METHOD SetDynConstraint_A : BOOL //Dynamic constraints for individual coordinates.
VAR_INPUT
    V : MC_LREAL; //equivalent to data type LREAL + MC_DEFAULT, MC_MAXIMUM
    A : MC_LREAL; //equivalent to data type LREAL + MC_DEFAULT, MC_MAXIMUM
    D : MC_LREAL; //equivalent to data type LREAL + MC_DEFAULT, MC_MAXIMUM
    J : MC_LREAL; //equivalent to data type LREAL + MC_DEFAULT, MC_MAXIMUM
END_VAR
THIS^.fbDynConstraintCoordinates.SetLimit(	Coordinate := Coord_Mcs_A1, 
											V := V, 
											A := A, 
											D := D, 
											J := J);
											
//Changes to the origin constraint do not affect the copy of the constraint in the instance of the DynamicConstraint_Container.
//For this reason, the container is being refreshed here							
fbDynConstraintContainer.Clear();
fbDynConstraintContainer.AddConstraint(fbDynConstraintPath);
fbDynConstraintContainer.AddConstraint(fbDynConstraintCoordinates);
END_METHOD

METHOD SetDynConstraint_B : BOOL //Dynamic constraints for individual coordinates.
VAR_INPUT
    V : MC_LREAL; //equivalent to data type LREAL + MC_DEFAULT, MC_MAXIMUM
    A : MC_LREAL; //equivalent to data type LREAL + MC_DEFAULT, MC_MAXIMUM
    D : MC_LREAL; //equivalent to data type LREAL + MC_DEFAULT, MC_MAXIMUM
    J : MC_LREAL; //equivalent to data type LREAL + MC_DEFAULT, MC_MAXIMUM
END_VAR
THIS^.fbDynConstraintCoordinates.SetLimit(	Coordinate := Coord_Mcs_B1, 
											V := V, 
											A := A, 
											D := D, 
											J := J);											

//Changes to the origin constraint do not affect the copy of the constraint in the instance of the DynamicConstraint_Container.
//For this reason, the container is being refreshed here							
fbDynConstraintContainer.Clear();
fbDynConstraintContainer.AddConstraint(fbDynConstraintPath);
fbDynConstraintContainer.AddConstraint(fbDynConstraintCoordinates);
END_METHOD

METHOD SetDynConstraint_C : BOOL //Dynamic constraints for individual coordinates.
VAR_INPUT
    V : MC_LREAL; //equivalent to data type LREAL + MC_DEFAULT, MC_MAXIMUM
    A : MC_LREAL; //equivalent to data type LREAL + MC_DEFAULT, MC_MAXIMUM
    D : MC_LREAL; //equivalent to data type LREAL + MC_DEFAULT, MC_MAXIMUM
    J : MC_LREAL; //equivalent to data type LREAL + MC_DEFAULT, MC_MAXIMUM
END_VAR
THIS^.fbDynConstraintCoordinates.SetLimit(	Coordinate := Coord_Mcs_C1, 
											V := V, 
											A := A, 
											D := D, 
											J := J);											

//Changes to the origin constraint do not affect the copy of the constraint in the instance of the DynamicConstraint_Container.
//For this reason, the container is being refreshed here							
fbDynConstraintContainer.Clear();
fbDynConstraintContainer.AddConstraint(fbDynConstraintPath);
fbDynConstraintContainer.AddConstraint(fbDynConstraintCoordinates);
END_METHOD

METHOD SetDynConstraint_Path : BOOL //One dimensional dynamic constraint along the XY-components of a path, ignoring non-tangential effects.
VAR_INPUT
    V : MC_LREAL; //equivalent to data type LREAL + MC_DEFAULT, MC_MAXIMUM
    A : MC_LREAL; //equivalent to data type LREAL + MC_DEFAULT, MC_MAXIMUM
    D : MC_LREAL; //equivalent to data type LREAL + MC_DEFAULT, MC_MAXIMUM
    J : MC_LREAL; //equivalent to data type LREAL + MC_DEFAULT, MC_MAXIMUM
END_VAR
THIS^.fbDynConstraintPath.SetValuesVADJ(V := V, 
										A := A, 
										D := D, 
										J := J);											

//Changes to the origin constraint do not affect the copy of the constraint in the instance of the DynamicConstraint_Container.
//For this reason, the container is being refreshed here							
fbDynConstraintContainer.Clear();
fbDynConstraintContainer.AddConstraint(fbDynConstraintPath);
fbDynConstraintContainer.AddConstraint(fbDynConstraintCoordinates);
END_METHOD

METHOD SetDynConstraint_X : BOOL //Dynamic constraints for individual coordinates.
VAR_INPUT
    V : MC_LREAL; //equivalent to data type LREAL + MC_DEFAULT, MC_MAXIMUM
    A : MC_LREAL; //equivalent to data type LREAL + MC_DEFAULT, MC_MAXIMUM
    D : MC_LREAL; //equivalent to data type LREAL + MC_DEFAULT, MC_MAXIMUM
    J : MC_LREAL; //equivalent to data type LREAL + MC_DEFAULT, MC_MAXIMUM
END_VAR
THIS^.fbDynConstraintCoordinates.SetLimit(	Coordinate := Coord_Mcs_X, 
											V := V, 
											A := A, 
											D := D, 
											J := J);											

//Changes to the origin constraint do not affect the copy of the constraint in the instance of the DynamicConstraint_Container.
//For this reason, the container is being refreshed here							
fbDynConstraintContainer.Clear();
fbDynConstraintContainer.AddConstraint(fbDynConstraintPath);
fbDynConstraintContainer.AddConstraint(fbDynConstraintCoordinates);
END_METHOD

METHOD SetDynConstraint_Y : BOOL //Dynamic constraints for individual coordinates.
VAR_INPUT
    V : MC_LREAL; //equivalent to data type LREAL + MC_DEFAULT, MC_MAXIMUM
    A : MC_LREAL; //equivalent to data type LREAL + MC_DEFAULT, MC_MAXIMUM
    D : MC_LREAL; //equivalent to data type LREAL + MC_DEFAULT, MC_MAXIMUM
    J : MC_LREAL; //equivalent to data type LREAL + MC_DEFAULT, MC_MAXIMUM
END_VAR
THIS^.fbDynConstraintCoordinates.SetLimit(	Coordinate := Coord_Mcs_Y, 
											V := V, 
											A := A, 
											D := D, 
											J := J);											

//Changes to the origin constraint do not affect the copy of the constraint in the instance of the DynamicConstraint_Container.
//For this reason, the container is being refreshed here							
fbDynConstraintContainer.Clear();
fbDynConstraintContainer.AddConstraint(fbDynConstraintPath);
fbDynConstraintContainer.AddConstraint(fbDynConstraintCoordinates);
END_METHOD

METHOD SetDynConstraint_Z : BOOL //Dynamic constraints for individual coordinates.
VAR_INPUT
    V : MC_LREAL; //equivalent to data type LREAL + MC_DEFAULT, MC_MAXIMUM
    A : MC_LREAL; //equivalent to data type LREAL + MC_DEFAULT, MC_MAXIMUM
    D : MC_LREAL; //equivalent to data type LREAL + MC_DEFAULT, MC_MAXIMUM
    J : MC_LREAL; //equivalent to data type LREAL + MC_DEFAULT, MC_MAXIMUM
END_VAR
THIS^.fbDynConstraintCoordinates.SetLimit(	Coordinate := Coord_Mcs_Z, 
											V := MC_DEFAULT, 
											A := A, 
											D := D, 
											J := J);											

//Changes to the origin constraint do not affect the copy of the constraint in the instance of the DynamicConstraint_Container.
//For this reason, the container is being refreshed here							
fbDynConstraintContainer.Clear();
fbDynConstraintContainer.AddConstraint(fbDynConstraintPath);
fbDynConstraintContainer.AddConstraint(fbDynConstraintCoordinates);
END_METHOD

METHOD Disable : HRESULT
VAR_INPUT
END_VAR
THIS^.eActiveCommand 				:= CHALET_NC.E_NcAxisCommands.Disable;
THIS^.fbFeedback.ActiveCommand 		:= TO_STRING(THIS^.eActiveCommand);	
THIS^.fbFeedback.LastCommandAccepted:= TRUE;		
THIS^.fbFeedback.Busy 				:= TRUE;

//Disable Axis
THIS^.fbMover.Disable(THIS^.fbFeedbackDisable);
Disable := S_OK;
END_METHOD

//This method is called when the system is disabled. Links are deleted as they may no longer be valid
METHOD Disassemble : HRESULT
VAR_INPUT
END_VAR

//Todo zzz Braucht es diese methode noch?
fbRouteComplete.Clear(); 
fbRouteRemaining.Clear(); 


Disassemble := S_OK;
END_METHOD

METHOD Enable : HRESULT
VAR_INPUT
END_VAR
IF NOT THIS^.fbFeedback.Busy THEN
	THIS^.eActiveCommand 				:= CHALET_NC.E_NcAxisCommands.Enable;
	THIS^.fbFeedback.ActiveCommand 		:= TO_STRING(THIS^.eActiveCommand);	
	THIS^.fbFeedback.LastCommandAccepted:= TRUE;		
	THIS^.fbFeedback.Busy 				:= TRUE;

	THIS^.fbMover.Enable(fbFeedbackEnable);
	Enable := S_OK;
ELSE
	Enable := S_FALSE;
	THIS^.fbFeedback.LastCommandAccepted:= FALSE;	
END_IF
END_METHOD

METHOD Reset : HRESULT
VAR_INPUT
END_VAR
THIS^.eActiveCommand 				:= CHALET_NC.E_NcAxisCommands.Reset;
THIS^.fbFeedback.ActiveCommand 		:= TO_STRING(THIS^.eActiveCommand);	
THIS^.fbFeedback.LastCommandAccepted:= TRUE;		
THIS^.fbFeedback.Busy 				:= TRUE;

THIS^.fbMover.Reset(THIS^.fbFeedbackReset);
Reset := S_OK;
END_METHOD

//Save the master mover and apply the distance traveled as a relative offset to this slave mover. Requires .StartExternalSetpoint()
METHOD AddMoverExtSetpoint : HRESULT
VAR_INPUT
	ipMasterMover : I_XP_Mover;
	fScalingX, fScalingY, fScalingZ, fScalingA, fScalingB, fScalingC : LREAL;// If >0, follow this axis to master-mover
END_VAR
//Invalide input
IF ipMasterMover = 0 THEN
	AddMoverExtSetpoint := E_FAIL;
	RETURN;
END_IF

//Allready stored a master
IF THIS^.ipMasterMover <> 0 THEN
	AddMoverExtSetpoint := E_FAIL;
	RETURN;
END_IF

//Only possible if ExternalSetpoint is not running
IF THIS^.nSeqStartExternalSetpoint <> 0 THEN
	AddMoverExtSetpoint := E_FAIL;
	RETURN;
END_IF



THIS^.ipMasterMover := ipMasterMover;
THIS^.stMasterMovementScaling.x := fScalingX;
THIS^.stMasterMovementScaling.y := fScalingy;
THIS^.stMasterMovementScaling.z := fScalingz;
THIS^.stMasterMovementScaling.a := fScalinga;
THIS^.stMasterMovementScaling.b := fScalingb;
THIS^.stMasterMovementScaling.c := fScalingc;
END_METHOD

{attribute 'monitoring':='call'}
PROPERTY  AxisExtSetpointA : CHALET_Nc.I_NcAxis_PLC
GET
AxisExtSetpointA := THIS^.AxisSetpointA;
END_GET
END_PROPERTY

{attribute 'monitoring':='call'}
PROPERTY AxisExtSetpointB : CHALET_Nc.I_NcAxis_PLC
GET
AxisExtSetpointB := THIS^.AxisSetpointB;
END_GET
END_PROPERTY

{attribute 'monitoring':='call'}
PROPERTY AxisExtSetpointC : CHALET_Nc.I_NcAxis_PLC
GET
AxisExtSetpointC := THIS^.AxisSetpointC;
END_GET
END_PROPERTY

{attribute 'monitoring':='call'}
PROPERTY  AxisExtSetpointX : CHALET_Nc.I_NcAxis_PLC
GET
AxisExtSetpointX := THIS^.AxisSetpointX;
END_GET
END_PROPERTY

{attribute 'monitoring':='call'}
PROPERTY AxisExtSetpointY : CHALET_Nc.I_NcAxis_PLC
GET
AxisExtSetpointY := THIS^.AxisSetpointY;
END_GET
END_PROPERTY

{attribute 'monitoring':='call'}
PROPERTY AxisExtSetpointZ : CHALET_Nc.I_NcAxis_PLC
GET
AxisExtSetpointZ := THIS^.AxisSetpointZ;
END_GET
END_PROPERTY

METHOD StartExternalSetpoint : HRESULT
THIS^.eActiveCommand 				:= CHALET_NC.E_NcAxisCommands.StartExternalSetpoint;
THIS^.fbFeedback.ActiveCommand 		:= TO_STRING(THIS^.eActiveCommand);		
THIS^.fbFeedback.Busy 				:= TRUE;


IF THIS^.fbMover.MCTOPLC.STD.State <> MC_PLANAR_STATE.Enabled THEN
	//Error wrong state
	
	;//zzz Todo Error message

ELSIF THIS^.bFeedExternalSetpointActive AND THIS^.nSeqStartExternalSetpoint = 999 THEN
	//Do nothing, setpoint is already active	
	THIS^.fbFeedbackExternalSetpointStartSeq.Done		:= TRUE;
	
ELSE
	
	//Start of internal sequence
	THIS^.fbFeedbackExternalSetpointStartSeq.Busy		:= TRUE;
	THIS^.nSeqStartExternalSetpoint := 1;
END_IF



StartExternalSetpoint := S_OK;
END_METHOD

METHOD StopExternalSetpoint : HRESULT
VAR_INPUT
END_VAR
AxisSetpointX.PowerOff();
AxisSetpointY.PowerOff();
AxisSetpointZ.PowerOff();
AxisSetpointA.PowerOff();
AxisSetpointB.PowerOff();
AxisSetpointC.PowerOff();


THIS^.eActiveCommand 				:= CHALET_NC.E_NcAxisCommands.StopExternalSetpoint;
THIS^.fbFeedback.ActiveCommand 		:= TO_STRING(THIS^.eActiveCommand);	
THIS^.fbFeedback.LastCommandAccepted:= TRUE;		


//Reset some flags
THIS^.nSeqStartExternalSetpoint := 0;
THIS^.bEvaluateFeedback := FALSE;
THIS^.ipMasterMover := 0;

IF THIS^.bFeedExternalSetpointActive THEN
	THIS^.fbMover.StopExternalSetpointGeneration(THIS^.fbFeedbackExtStop);	
	THIS^.bFeedExternalSetpointActive 	:= FALSE;
	THIS^.fbFeedback.Busy 				:= TRUE;
ELSE
	THIS^.fbFeedback.Done 				:= TRUE;
END_IF


StopExternalSetpoint := S_OK;
END_METHOD

METHOD PROTECTED UpdateExternalSetpoint : HRESULT
VAR
	SetPos, SetVelo, SetAcc : MoverVector;
	hr : HRESULT;
	stStartOptions : ST_ExternalSetpointGenerationOptions;
	stPosDifferenceToMasterMover : MoverVector;
	stPosOffsetMasterMover : MoverVector;
	stVeloOffsetMasterMover : MoverVector;
	stAccOffsetMasterMover : MoverVector;
END_VAR
IF NOT THIS^.Enabled THEN
	THIS^.nSeqStartExternalSetpoint := 0;
	THIS^.bFeedExternalSetpointActive := FALSE;
	THIS^.bEvaluateFeedback := FALSE;
END_IF


CASE nSeqStartExternalSetpoint OF
	0: //Wait for start
		;
		
	1: 	//store position of Master-Mover
		IF (THIS^.ipMasterMover <> 0) THEN
			THIS^.stMasterPositionAtStart := THIS^.ipMasterMover.PositionSet;
		END_IF

		//Reset all axis
		IF AxisSetpointX.Mapped THEN
			AxisSetpointX.Reset();
		END_IF
		IF AxisSetpointY.Mapped THEN
			AxisSetpointY.Reset();
		END_IF
		IF AxisSetpointZ.Mapped THEN
			AxisSetpointZ.Reset();
		END_IF
		IF AxisSetpointA.Mapped THEN
			AxisSetpointA.Reset();
		END_IF
		IF AxisSetpointB.Mapped THEN
			AxisSetpointB.Reset();
		END_IF
		IF AxisSetpointC.Mapped THEN
			AxisSetpointC.Reset();
		END_IF
		nSeqStartExternalSetpoint := nSeqStartExternalSetpoint + 1;		
		
		
	2: //Wait for feedback
		IF AxisSetpointX.Mapped THEN hr := GetMostSignificant(hr, AxisSetpointX.Feedback.HR); END_IF
		IF AxisSetpointY.Mapped THEN hr := GetMostSignificant(hr, AxisSetpointY.Feedback.HR); END_IF
		IF AxisSetpointZ.Mapped THEN hr := GetMostSignificant(hr, AxisSetpointZ.Feedback.HR); END_IF
		IF AxisSetpointA.Mapped THEN hr := GetMostSignificant(hr, AxisSetpointA.Feedback.HR); END_IF
		IF AxisSetpointB.Mapped THEN hr := GetMostSignificant(hr, AxisSetpointB.Feedback.HR); END_IF
		IF AxisSetpointC.Mapped THEN hr := GetMostSignificant(hr, AxisSetpointC.Feedback.HR); END_IF	
		IF hr = S_OK THEN
		 	nSeqStartExternalSetpoint := nSeqStartExternalSetpoint + 1;	
		END_IF
		
	3: 	//Reset all axis
		IF AxisSetpointX.Mapped THEN
			AxisSetpointX.PowerOn();
		END_IF
		IF AxisSetpointY.Mapped THEN
			AxisSetpointY.PowerOn();
		END_IF
		IF AxisSetpointZ.Mapped THEN
			AxisSetpointZ.PowerOn();
		END_IF
		IF AxisSetpointA.Mapped THEN
			AxisSetpointA.PowerOn();
		END_IF
		IF AxisSetpointB.Mapped THEN
			AxisSetpointB.PowerOn();
		END_IF
		IF AxisSetpointC.Mapped THEN
			AxisSetpointC.PowerOn();
		END_IF
		nSeqStartExternalSetpoint := nSeqStartExternalSetpoint + 1;		
		
	4: //Wait for feedback
		IF AxisSetpointX.Mapped THEN hr := GetMostSignificant(hr, AxisSetpointX.Feedback.HR); END_IF
		IF AxisSetpointY.Mapped THEN hr := GetMostSignificant(hr, AxisSetpointY.Feedback.HR); END_IF
		IF AxisSetpointZ.Mapped THEN hr := GetMostSignificant(hr, AxisSetpointZ.Feedback.HR); END_IF
		IF AxisSetpointA.Mapped THEN hr := GetMostSignificant(hr, AxisSetpointA.Feedback.HR); END_IF
		IF AxisSetpointB.Mapped THEN hr := GetMostSignificant(hr, AxisSetpointB.Feedback.HR); END_IF
		IF AxisSetpointC.Mapped THEN hr := GetMostSignificant(hr, AxisSetpointC.Feedback.HR); END_IF	
		IF hr = S_OK THEN
		 	nSeqStartExternalSetpoint := nSeqStartExternalSetpoint + 1;	
		END_IF

	5: 	//Enable all axis
		IF AxisSetpointX.Mapped THEN
			AxisSetpointX.SetActPosition(0.0);
		END_IF
		IF AxisSetpointY.Mapped THEN
			AxisSetpointY.SetActPosition(0.0);
		END_IF
		IF AxisSetpointZ.Mapped THEN
			AxisSetpointZ.SetActPosition(0.0);
		END_IF
		IF AxisSetpointA.Mapped THEN
			AxisSetpointA.SetActPosition(0.0);
		END_IF
		IF AxisSetpointB.Mapped THEN
			AxisSetpointB.SetActPosition(0.0);
		END_IF
		IF AxisSetpointC.Mapped THEN
			AxisSetpointC.SetActPosition(0.0);
		END_IF
		nSeqStartExternalSetpoint := nSeqStartExternalSetpoint + 1;		
		
	6: //Wait for feedback
		IF AxisSetpointX.Mapped THEN hr := GetMostSignificant(hr, AxisSetpointX.Feedback.HR); END_IF
		IF AxisSetpointY.Mapped THEN hr := GetMostSignificant(hr, AxisSetpointY.Feedback.HR); END_IF
		IF AxisSetpointZ.Mapped THEN hr := GetMostSignificant(hr, AxisSetpointZ.Feedback.HR); END_IF
		IF AxisSetpointA.Mapped THEN hr := GetMostSignificant(hr, AxisSetpointA.Feedback.HR); END_IF
		IF AxisSetpointB.Mapped THEN hr := GetMostSignificant(hr, AxisSetpointB.Feedback.HR); END_IF
		IF AxisSetpointC.Mapped THEN hr := GetMostSignificant(hr, AxisSetpointC.Feedback.HR); END_IF	
		IF hr = S_OK THEN
		 	nSeqStartExternalSetpoint := nSeqStartExternalSetpoint + 1;	
		END_IF

		
	7: // Activate external setpoint mode on mover
		stStartOptions.Mode := MC_EXTERNAL_SET_POSITION_MODE.Relative;
		THIS^.fbMover.StartExternalSetpointGeneration(	commandFeedback	:= THIS^.fbFeedbackExtStart,
														options 		:= stStartOptions);
		THIS^.bFeedExternalSetpointActive := TRUE;												
		nSeqStartExternalSetpoint := nSeqStartExternalSetpoint + 1;
	
		
	8: 
		THIS^.bEvaluateFeedback := TRUE;
		IF THIS^.fbFeedbackExtStart.Done THEN
			//Finish Sequence
			fbFeedbackExternalSetpointStartSeq.Done := TRUE;
			nSeqStartExternalSetpoint := 999;
		END_IF
		
	999: // finish seqence feedback
		
		
	1000..1999:
		//Error
		fbFeedbackExternalSetpointStartSeq.HR := E_FAIL;
END_CASE



IF THIS^.bFeedExternalSetpointActive THEN
	SetPos.X := AxisSetpointX.SetPosition;
	SetPos.Y := AxisSetpointY.SetPosition;
	SetPos.Z := AxisSetpointZ.SetPosition;
	SetPos.A := AxisSetpointA.SetPosition;
	SetPos.B := AxisSetpointB.SetPosition;
	SetPos.C := AxisSetpointC.SetPosition;
	
	SetVelo.X := AxisSetpointX.SetVelocity;
	SetVelo.Y := AxisSetpointY.SetVelocity;
	SetVelo.Z := AxisSetpointZ.SetVelocity;
	SetVelo.A := AxisSetpointA.SetVelocity;
	SetVelo.B := AxisSetpointB.SetVelocity;
	SetVelo.C := AxisSetpointC.SetVelocity;
	
	SetAcc.X := AxisSetpointX.SetAcceleration;
	SetAcc.Y := AxisSetpointY.SetAcceleration;
	SetAcc.Z := AxisSetpointZ.SetAcceleration;
	SetAcc.A := AxisSetpointA.SetAcceleration;
	SetAcc.B := AxisSetpointB.SetAcceleration;
	SetAcc.C := AxisSetpointC.SetAcceleration;
	
	IF THIS^.ipMasterMover <> 0 THEN
		//Difference to gearIn position
		stPosDifferenceToMasterMover := F_Vector_Subtraction(	minuend := THIS^.ipMasterMover.PositionSet, 
																subtrahend := stMasterPositionAtStart);
		//Add scaling factor	
		stPosOffsetMasterMover := F_Vector_Multiplication(	factor1 := stPosDifferenceToMasterMover,
															factor2 := THIS^.stMasterMovementScaling);							
		stVeloOffsetMasterMover := F_Vector_Multiplication(	factor1 := THIS^.ipMasterMover.VelocitySet,
															factor2 := THIS^.stMasterMovementScaling);							
		stAccOffsetMasterMover := F_Vector_Multiplication(	factor1 := THIS^.ipMasterMover.AccelerationSet,
															factor2 := THIS^.stMasterMovementScaling);						
		
		
		//Add Mastermover-Offest to 6-Axis-Offset
		SetPos := F_Vector_Addition( 	summand1 := stPosOffsetMasterMover,
									 	summand2 := SetPos);
		SetVelo := F_Vector_Addition( 	summand1 := stVeloOffsetMasterMover,
									 	summand2 := SetVelo);
		SetAcc := F_Vector_Addition( 	summand1 := stAccOffsetMasterMover,
									 	summand2 := SetAcc);
														
	END_IF
	
	//Send data to mover
	THIS^.fbMover.SetExternalSetpoint(	setPosition 		:= SetPos, 
										setVelocity 		:= SetVelo,
										setAcceleration 	:= SetAcc);
END_IF



CASE THIS^.eActiveCommand OF
	//Add the 6 axis to the feedback			
	E_NcAxisCommands.StartExternalSetpoint:
		//Only check MC_PlanarFeedback if cmd is active. Ignore old feedback
		IF THIS^.bEvaluateFeedback THEN
			fbFeedback.Busy 		:= fbFeedbackExtStart.Busy;
			fbFeedback.Done 		:= fbFeedbackExtStart.Done;
			fbFeedback.ErrorId 		:= fbFeedbackExtStart.ErrorID;
			fbFeedback.ClearObjectInfo();
		END_IF
		fbFeedback.HR := GetMostSignificant(fbFeedback.HR, fbFeedbackExternalSetpointStartSeq.HR);
		IF AxisSetpointX.Mapped THEN fbFeedback.HR := GetMostSignificant(fbFeedback.HR, AxisSetpointX.Feedback.HR);END_IF
		IF AxisSetpointY.Mapped THEN fbFeedback.HR := GetMostSignificant(fbFeedback.HR, AxisSetpointY.Feedback.HR);END_IF
		IF AxisSetpointZ.Mapped THEN fbFeedback.HR := GetMostSignificant(fbFeedback.HR, AxisSetpointZ.Feedback.HR);END_IF
		IF AxisSetpointA.Mapped THEN fbFeedback.HR := GetMostSignificant(fbFeedback.HR, AxisSetpointA.Feedback.HR);END_IF
		IF AxisSetpointB.Mapped THEN fbFeedback.HR := GetMostSignificant(fbFeedback.HR, AxisSetpointB.Feedback.HR);END_IF
		IF AxisSetpointC.Mapped THEN fbFeedback.HR := GetMostSignificant(fbFeedback.HR, AxisSetpointC.Feedback.HR);END_IF
		
	//Add the 6 axis to the feedback	
	E_NcAxisCommands.StopExternalSetpoint:
		fbFeedback.Busy 		:= fbFeedbackExtStop.Busy;
		fbFeedback.Done 		:= fbFeedbackExtStop.Done;
		fbFeedback.ErrorId 		:= fbFeedbackExtStop.ErrorID;
		fbFeedback.ClearObjectInfo(); 
		IF AxisSetpointX.Mapped THEN fbFeedback.HR := GetMostSignificant(fbFeedback.HR, AxisSetpointX.Feedback.HR);END_IF
		IF AxisSetpointY.Mapped THEN fbFeedback.HR := GetMostSignificant(fbFeedback.HR, AxisSetpointY.Feedback.HR);END_IF
		IF AxisSetpointZ.Mapped THEN fbFeedback.HR := GetMostSignificant(fbFeedback.HR, AxisSetpointZ.Feedback.HR);END_IF
		IF AxisSetpointA.Mapped THEN fbFeedback.HR := GetMostSignificant(fbFeedback.HR, AxisSetpointA.Feedback.HR);END_IF
		IF AxisSetpointB.Mapped THEN fbFeedback.HR := GetMostSignificant(fbFeedback.HR, AxisSetpointB.Feedback.HR);END_IF
		IF AxisSetpointC.Mapped THEN fbFeedback.HR := GetMostSignificant(fbFeedback.HR, AxisSetpointC.Feedback.HR);END_IF
END_CASE		


fbFeedbackExtStart.Update(); 
fbFeedbackExtStop.Update(); 


IF AxisSetpointX.Mapped THEN AxisSetpointX.Update() ;END_IF
IF AxisSetpointY.Mapped THEN AxisSetpointY.Update() ;END_IF
IF AxisSetpointZ.Mapped THEN AxisSetpointZ.Update() ;END_IF
IF AxisSetpointA.Mapped THEN AxisSetpointA.Update() ;END_IF
IF AxisSetpointB.Mapped THEN AxisSetpointB.Update() ;END_IF
IF AxisSetpointC.Mapped THEN AxisSetpointC.Update() ;END_IF
END_METHOD

METHOD AddToGroup : HRESULT
VAR_INPUT
	iGroup : I_XP_Group;
END_VAR
IF NOT THIS^.fbFeedback.Busy THEN
	THIS^.eActiveCommand 				:= CHALET_NC.E_NcAxisCommands.AddToGroupe;
	THIS^.fbFeedback.ActiveCommand 		:= TO_STRING(THIS^.eActiveCommand);	
	THIS^.fbFeedback.LastCommandAccepted:= TRUE;		
	THIS^.fbFeedback.Busy 				:= TRUE;
	
	iGroup.AddMover(THIS^.fbMover, THIS^.fbFeedbackAddToGrp);
	AddToGroup := S_OK;
ELSE
	AddToGroup := S_FALSE;
	THIS^.fbFeedback.LastCommandAccepted:= FALSE;	
END_IF
END_METHOD

METHOD RemoveFromGroup : HRESULT

VAR
	iGroup: INT;
END_VAR
IF NOT THIS^.fbFeedback.Busy THEN
	THIS^.eActiveCommand 				:= CHALET_NC.E_NcAxisCommands.RemoveFromGroupe;
	THIS^.fbFeedback.ActiveCommand 	:= TO_STRING(THIS^.eActiveCommand);	
	THIS^.fbFeedback.LastCommandAccepted:= TRUE;		
	THIS^.fbFeedback.Busy 				:= TRUE;
	
	THIS^.fbMover.RemoveFromGroup(THIS^.fbFeedbackRmvFromGrp);
	
	RemoveFromGroup := S_OK;
ELSE
	RemoveFromGroup := S_FALSE;
	THIS^.fbFeedback.LastCommandAccepted:= FALSE;	
END_IF
END_METHOD

//The mover returns to its SetPos. The force of the Z, A and B axis is slowly increased.
METHOD LiftFromUnknownLevel : HRESULT
VAR_INPUT
END_VAR
THIS^.eActiveCommand 				:= CHALET_NC.E_NcAxisCommands.LiftFromUnknownLevel;
THIS^.fbFeedback.ActiveCommand 		:= TO_STRING(THIS^.eActiveCommand);		
THIS^.fbFeedback.Busy 				:= TRUE;


IF THIS^.fbMover.MCTOPLC.STD.State <> MC_PLANAR_STATE.Enabled THEN
	//Error wrong state
	
	;//zzz Todo Error message
	
ELSIF NOT THIS^.Standstill THEN
	//Error not allowed if mover is moving
	
	;//zzz Todo Error message
	
ELSE
	//Start of internal sequence
	THIS^.fbFeedbackLiftFromUnknown.Busy		:= TRUE;
	THIS^.nSeqLiftFromUnknown := 1;
	THIS^.nSeqLowerToUnknown := 0;
END_IF



LiftFromUnknownLevel := S_OK;
END_METHOD

(* The mover is lowered. The target height is unknown. The force from the Z, A and B axles is then reduced to a minimum. X, Y and C still remain active.
   This function can be used, for example, to place the mover in a holder.  *)
METHOD LowerToUnknownLevel : HRESULT
VAR_INPUT
END_VAR
THIS^.eActiveCommand 				:= CHALET_NC.E_NcAxisCommands.LowerToUnknownLevel;
THIS^.fbFeedback.ActiveCommand 		:= TO_STRING(THIS^.eActiveCommand);		
THIS^.fbFeedback.Busy 				:= TRUE;


IF THIS^.fbMover.MCTOPLC.STD.State <> MC_PLANAR_STATE.Enabled THEN
	//Error wrong state
	
	;//zzz Todo Error message

ELSIF NOT THIS^.Standstill THEN
	//Error not allowed if mover is moving
	
	;//zzz Todo Error message
	
	
ELSE
	//Start of internal sequence
	THIS^.fbFeedbackLowerToUnknown.Busy		:= TRUE;
	THIS^.nSeqLowerToUnknown := 1;
	THIS^.nSeqLiftFromUnknown := 0;
END_IF



LowerToUnknownLevel := S_OK;
END_METHOD

METHOD PROTECTED UpdateUnknownLevel : HRESULT
VAR
	hr : HRESULT;
	stForceLimitMax: Tc3_XPlanarUtility.Force6D;
	stForceLimitMin: Tc3_XPlanarUtility.Force6D;
	stPosLagValueTemp : MoverVector;
	ipComObject: Tc3_Module.ITComObject;
	pstForcesAtBeginn : POINTER TO MoverVector;
END_VAR
VAR_INST
	fLowerNPerS : LREAL := 30.0;
	fLiftNPerS : LREAL := 50.0;
	fMaxForceFactor : LREAL := 1.0;
	fMinForceFactor : LREAL := 0.1;
	fPowerFactor : LREAL := 1.0;
	fCycleTime_s : LREAL; //[s]	
	bDoOnceIfDisabled : BOOL;
	stLagValuesAtBeginn : MoverVector;
	stForcesAtBeginn :  MoverVector;
	stForceLimitMaxAtBeginn : Tc3_XPlanarUtility.Force6D;
	stForceLimitMinAtBeginn : Tc3_XPlanarUtility.Force6D;
	stValideMinForce		: Tc3_XPlanarUtility.Force6D;
END_VAR
VAR CONSTANT
	N_PTCID_ForceLimitMax : PTCID := 16#03175051;
	N_PTCID_ForceLimitMin : PTCID := 16#03175052;
END_VAR
IF NOT THIS^.Enabled THEN
	THIS^.nSeqLowerToUnknown := 0;
	THIS^.nSeqLiftFromUnknown := 0;
	
	fCycleTime_s :=  TO_LREAL(TwinCAT_SystemInfoVarList._TaskInfo[THIS^.nTaskIndex].CycleTime(*100ns*)) / 10_000_000.0;
	stLagValuesAtBeginn := THIS^.UtilityMcMover.GetMaximumPositionLagValue();
END_IF

//if no TcIoMover is linked e.g. MC-Mover is in Simulation Mover:
IF THIS^.UtilityTcIoMover = 0 THEN
	IF fbFeedbackLowerToUnknown.Busy THEN
		fbFeedbackLowerToUnknown.Done := TRUE;
	END_IF
	IF fbFeedbackLiftFromUnknown.Busy THEN
		fbFeedbackLiftFromUnknown.Done := TRUE;
	END_IF
	RETURN;
END_IF



IF THIS^.ipXpSystem.Disabled AND bDoOnceIfDisabled THEN
	bDoOnceIfDisabled := FALSE;
	fPowerFactor := fMaxForceFactor;
	
	FW_ObjMgr_GetObjectInstance(oid:= THIS^.UtilityTcIoMover.ObjectId, iid:= TC_GLOBAL_IID_LIST.IID_ITComObject, pipUnk:= ADR(ipComObject));
	IF ipComObject <> 0 THEN
		// No minimum can be set if one of the 6 values in the struct is greater than the maximum. Equal is allowed.
		// The minimum is therefore first written to something valid. Followed by Max and the original minimum
		hr := ipComObject.TcSetObjPara(pid := N_PTCID_ForceLimitMin, nData := SIZEOF(stValideMinForce), pData := ADR(stValideMinForce), pgp := 0);
		hr := ipComObject.TcSetObjPara(pid := N_PTCID_ForceLimitMax, nData := SIZEOF(stForceLimitMaxAtBeginn), pData := ADR(stForceLimitMaxAtBeginn), pgp := 0);
		hr := ipComObject.TcSetObjPara(pid := N_PTCID_ForceLimitMin, nData := SIZEOF(stForceLimitMinAtBeginn), pData := ADR(stForceLimitMinAtBeginn), pgp := 0);
		FW_SafeRelease(ADR(ipComObject));
	END_IF

	THIS^.UtilityMcMover.SetMaximumPositionLagValue(stLagValuesAtBeginn);
END_IF


//Down
CASE nSeqLowerToUnknown OF
	0: //Wait for start
		;
		
	1: // Check if not already lewered	
		IF fPowerFactor = fMinForceFactor THEN
			nSeqLowerToUnknown := 999;
		ELSE
			nSeqLowerToUnknown := 5;
		END_IF
		
	5:	//Get some values
		pstForcesAtBeginn := THIS^.UtilityTcIoMover.ScopeAdr.GetOutputForce();
		stForcesAtBeginn := pstForcesAtBeginn^;
		stForceLimitMaxAtBeginn := THIS^.UtilityTcIoMover.GetForceLimitMax();
		stForceLimitMinAtBeginn := THIS^.UtilityTcIoMover.GetForceLimitMin();
		stValideMinForce.Fx := (stForceLimitMinAtBeginn.Fx * fMinForceFactor);
		stValideMinForce.Fy := (stForceLimitMinAtBeginn.Fy * fMinForceFactor);
		stValideMinForce.Fz := (stForceLimitMinAtBeginn.Fz * fMinForceFactor);
		stValideMinForce.Mx := (stForceLimitMinAtBeginn.Mx * fMinForceFactor);
		stValideMinForce.My := (stForceLimitMinAtBeginn.My * fMinForceFactor);
		stValideMinForce.Mz := (stForceLimitMinAtBeginn.Mz * fMinForceFactor);
		bDoOnceIfDisabled := TRUE;
		
		stPosLagValueTemp := stLagValuesAtBeginn;
		stPosLagValueTemp.z := THIS^.PositionSet.z + 0.5;
		THIS^.UtilityMcMover.SetMaximumPositionLagValue(stPosLagValueTemp);
		
		
		//0.0 - 1.0
		fPowerFactor := (stForcesAtBeginn.z / stForceLimitMaxAtBeginn.Fz);
		
		//add 5%
		fPowerFactor := fPowerFactor + 0.05;
		
		//Limit to 0.1 - 1.0
		fPowerFactor := MIN(fPowerFactor, fMaxForceFactor);
		fPowerFactor := MAX(fPowerFactor, fMinForceFactor);
		
		//set force Z, a and b
		stForceLimitMin := stForceLimitMinAtBeginn;		
		stForceLimitMin.fz := stForceLimitMin.Fz * fPowerFactor;
		stForceLimitMin.Mx := stForceLimitMin.Mx * fPowerFactor;
		stForceLimitMin.My := stForceLimitMin.My * fPowerFactor;
		
		stForceLimitMax := stForceLimitMaxAtBeginn;	
		stForceLimitMax.fz := stForceLimitMax.Fz * fPowerFactor;
		stForceLimitMax.Mx := stForceLimitMax.Mx * fPowerFactor;
		stForceLimitMax.My := stForceLimitMax.My * fPowerFactor;

		// 13.01.2025 Todo PLC Chash if Min > Max. use objParm insted
		//	THIS^.TcIoXPlanarMover.SetForceLimitMin(stForceLimitMin);
		//	THIS^.TcIoXPlanarMover.SetForceLimitMax(stForceLimitMax);
		FW_ObjMgr_GetObjectInstance(oid:= THIS^.UtilityTcIoMover.ObjectId, iid:= TC_GLOBAL_IID_LIST.IID_ITComObject, pipUnk:= ADR(ipComObject));
		IF ipComObject <> 0 THEN	
			// No minimum can be set if one of the 6 values in the struct is greater than the maximum. Equal is allowed.
			// The minimum is therefore first written to something valid. Followed by Max and the original minimum
			hr := ipComObject.TcSetObjPara(pid := N_PTCID_ForceLimitMin, nData := SIZEOF(stValideMinForce), pData := ADR(stValideMinForce), pgp := 0);
			hr := ipComObject.TcSetObjPara(pid := N_PTCID_ForceLimitMax, nData := SIZEOF(stForceLimitMax), pData := ADR(stForceLimitMax), pgp := 0);
			hr := ipComObject.TcSetObjPara(pid := N_PTCID_ForceLimitMin, nData := SIZEOF(stForceLimitMin), pData := ADR(stForceLimitMin), pgp := 0);
			FW_SafeRelease(ADR(ipComObject));
		END_IF

	
		nSeqLowerToUnknown := 10;
		
		
	10: 	
		//A lowering of the mover was detected followed by speed ~0
		IF (THIS^.PositionAct.z < THIS^.PositionSet.z * 0.5) AND (ABS(THIS^.VelocityAct.z) < 5.0)  THEN
			nSeqLowerToUnknown := 20;
			
		ELSIF (fPowerFactor <= fMinForceFactor) THEN
			nSeqLowerToUnknown := 20;
				
		ELSE
			//Reduce force each cycle
			fPowerFactor := fPowerFactor - ((fLowerNPerS/stForceLimitMaxAtBeginn.Fz) * fCycleTime_s);
					
			//Limit to 0.1 - 1.0
			fPowerFactor := MIN(fPowerFactor, fMaxForceFactor);
			fPowerFactor := MAX(fPowerFactor, fMinForceFactor);
			
			//set force Z, a and b to current + 10%
			stForceLimitMin := stForceLimitMinAtBeginn;		
			stForceLimitMin.fz := stForceLimitMin.Fz * fPowerFactor;
			stForceLimitMin.Mx := stForceLimitMin.Mx * fPowerFactor;
			stForceLimitMin.My := stForceLimitMin.My * fPowerFactor;
			
			stForceLimitMax := stForceLimitMaxAtBeginn;	
			stForceLimitMax.fz := stForceLimitMax.Fz * fPowerFactor;
			stForceLimitMax.Mx := stForceLimitMax.Mx * fPowerFactor;
			stForceLimitMax.My := stForceLimitMax.My * fPowerFactor;
	
			// 13.01.2025 Todo PLC Chash if Min > Max. use objParm insted
			//	THIS^.TcIoXPlanarMover.SetForceLimitMin(stForceLimitMin);
			//	THIS^.TcIoXPlanarMover.SetForceLimitMax(stForceLimitMax);
			FW_ObjMgr_GetObjectInstance(oid:= THIS^.UtilityTcIoMover.ObjectId, iid:= TC_GLOBAL_IID_LIST.IID_ITComObject, pipUnk:= ADR(ipComObject));
			IF ipComObject <> 0 THEN
				// No minimum can be set if one of the 6 values in the struct is greater than the maximum. Equal is allowed.
				// The minimum is therefore first written to something valid. Followed by Max and the original minimum
				hr := ipComObject.TcSetObjPara(pid := N_PTCID_ForceLimitMin, nData := SIZEOF(stValideMinForce), pData := ADR(stValideMinForce), pgp := 0);
				hr := ipComObject.TcSetObjPara(pid := N_PTCID_ForceLimitMax, nData := SIZEOF(stForceLimitMax), pData := ADR(stForceLimitMax), pgp := 0);
				hr := ipComObject.TcSetObjPara(pid := N_PTCID_ForceLimitMin, nData := SIZEOF(stForceLimitMin), pData := ADR(stForceLimitMin), pgp := 0);
				FW_SafeRelease(ADR(ipComObject));
			END_IF

	
		END_IF
	
		
	20: // Reduce Force to minimum
		fPowerFactor := fMinForceFactor;
		
		//set force Z, a and b to minimum
		stForceLimitMin := stForceLimitMinAtBeginn;		
		stForceLimitMin.fz := stForceLimitMin.Fz * fPowerFactor;
		stForceLimitMin.Mx := stForceLimitMin.Mx * fPowerFactor;
		stForceLimitMin.My := stForceLimitMin.My * fPowerFactor;
		
		stForceLimitMax := stForceLimitMaxAtBeginn;	
		stForceLimitMax.fz := stForceLimitMax.Fz * fPowerFactor;
		stForceLimitMax.Mx := stForceLimitMax.Mx * fPowerFactor;
		stForceLimitMax.My := stForceLimitMax.My * fPowerFactor;
	    
	    
		// 13.01.2025 Todo PLC Chash if Min > Max. use objParm insted
		//	THIS^.TcIoXPlanarMover.SetForceLimitMin(stForceLimitMin);
		//	THIS^.TcIoXPlanarMover.SetForceLimitMax(stForceLimitMax);
		FW_ObjMgr_GetObjectInstance(oid:= THIS^.UtilityTcIoMover.ObjectId, iid:= TC_GLOBAL_IID_LIST.IID_ITComObject, pipUnk:= ADR(ipComObject));
		IF ipComObject <> 0 THEN
			// No minimum can be set if one of the 6 values in the struct is greater than the maximum. Equal is allowed.
			// The minimum is therefore first written to something valid. Followed by Max and the original minimum
			hr := ipComObject.TcSetObjPara(pid := N_PTCID_ForceLimitMin, nData := SIZEOF(stValideMinForce), pData := ADR(stValideMinForce), pgp := 0);
			hr := ipComObject.TcSetObjPara(pid := N_PTCID_ForceLimitMax, nData := SIZEOF(stForceLimitMax), pData := ADR(stForceLimitMax), pgp := 0);
			hr := ipComObject.TcSetObjPara(pid := N_PTCID_ForceLimitMin, nData := SIZEOF(stForceLimitMin), pData := ADR(stForceLimitMin), pgp := 0);
			FW_SafeRelease(ADR(ipComObject));
		END_IF

		
		nSeqLowerToUnknown := 999;
				
	999: // finish seqence feedback
		fbFeedbackLowerToUnknown.Done := TRUE;
		
	1000..1999:
		//Error
		fbFeedbackLowerToUnknown.HR := E_FAIL;
END_CASE



//Up
CASE nSeqLiftFromUnknown OF
	0: //Wait for start
		;
		
	1: // Check if not already lifted	
		IF fPowerFactor = fMaxForceFactor THEN
			nSeqLiftFromUnknown := 999;
		ELSE
			nSeqLiftFromUnknown := 5;
		END_IF		
		
	5: 
		//0.0 - 1.0
		fPowerFactor := (stForcesAtBeginn.z / stForceLimitMaxAtBeginn.Fz);
		
		// -5%
		fPowerFactor := fPowerFactor - 0.05;
		
		//Limit to 0.1 - 1.0
		fPowerFactor := MIN(fPowerFactor, fMaxForceFactor);
		fPowerFactor := MAX(fPowerFactor, fMinForceFactor);
		
		//set force Z, a and b
		stForceLimitMin := stForceLimitMinAtBeginn;		
		stForceLimitMin.fz := stForceLimitMin.Fz * fPowerFactor;
		stForceLimitMin.Mx := stForceLimitMin.Mx * fPowerFactor;
		stForceLimitMin.My := stForceLimitMin.My * fPowerFactor;
		
		stForceLimitMax := stForceLimitMaxAtBeginn;	
		stForceLimitMax.fz := stForceLimitMax.Fz * fPowerFactor;
		stForceLimitMax.Mx := stForceLimitMax.Mx * fPowerFactor;
		stForceLimitMax.My := stForceLimitMax.My * fPowerFactor;

		// 13.01.2025 Todo PLC Chash if Min > Max. use objParm insted
		//THIS^.TcIoXPlanarMover.SetForceLimitMax(stForceLimitMax);
		//THIS^.TcIoXPlanarMover.SetForceLimitMin(stForceLimitMin);
		FW_ObjMgr_GetObjectInstance(oid:= THIS^.UtilityTcIoMover.ObjectId, iid:= TC_GLOBAL_IID_LIST.IID_ITComObject, pipUnk:= ADR(ipComObject));
		IF ipComObject <> 0 THEN
			// No minimum can be set if one of the 6 values in the struct is greater than the maximum. Equal is allowed.
			// The minimum is therefore first written to something valid. Followed by Max and the original minimum
			hr := ipComObject.TcSetObjPara(pid := N_PTCID_ForceLimitMin, nData := SIZEOF(stValideMinForce), pData := ADR(stValideMinForce), pgp := 0);
			hr := ipComObject.TcSetObjPara(pid := N_PTCID_ForceLimitMax, nData := SIZEOF(stForceLimitMax), pData := ADR(stForceLimitMax), pgp := 0);
			hr := ipComObject.TcSetObjPara(pid := N_PTCID_ForceLimitMin, nData := SIZEOF(stForceLimitMin), pData := ADR(stForceLimitMin), pgp := 0);
			FW_SafeRelease(ADR(ipComObject));
		END_IF
		
		nSeqLiftFromUnknown := 10;
		

		
	10: 	
		//A lift of the mover was detected followed by speed ~0
		IF (THIS^.PositionAct.z > THIS^.PositionSet.z * 0.5) AND (ABS(THIS^.VelocityAct.z) < 5.0)  THEN
			nSeqLiftFromUnknown := 20;
			
		ELSIF (fPowerFactor >= fMaxForceFactor ) THEN
			nSeqLiftFromUnknown := 20;
				
		ELSE
			//Reduce force each cycle
			fPowerFactor := fPowerFactor + ((fLiftNPerS/stForceLimitMaxAtBeginn.Fz) * fCycleTime_s);
					
			//Limit to 0.1 - 1.0
			fPowerFactor := MIN(fPowerFactor, fMaxForceFactor);
			fPowerFactor := MAX(fPowerFactor, fMinForceFactor);
			
			//set force Z, a and b 
			stForceLimitMin := stForceLimitMinAtBeginn;		
			stForceLimitMin.fz := stForceLimitMin.Fz * fPowerFactor;
			stForceLimitMin.Mx := stForceLimitMin.Mx * fPowerFactor;
			stForceLimitMin.My := stForceLimitMin.My * fPowerFactor;
			
			stForceLimitMax := stForceLimitMaxAtBeginn;	
			stForceLimitMax.fz := stForceLimitMax.Fz * fPowerFactor;
			stForceLimitMax.Mx := stForceLimitMax.Mx * fPowerFactor;
			stForceLimitMax.My := stForceLimitMax.My * fPowerFactor;
	
	
		// 13.01.2025 Todo PLC Chash if Min > Max. use objParm insted
		//THIS^.TcIoXPlanarMover.SetForceLimitMax(stForceLimitMax);
		//THIS^.TcIoXPlanarMover.SetForceLimitMin(stForceLimitMin);
		FW_ObjMgr_GetObjectInstance(oid:= THIS^.UtilityTcIoMover.ObjectId, iid:= TC_GLOBAL_IID_LIST.IID_ITComObject, pipUnk:= ADR(ipComObject));
		IF ipComObject <> 0 THEN
			// No minimum can be set if one of the 6 values in the struct is greater than the maximum. Equal is allowed.
			// The minimum is therefore first written to something valid. Followed by Max and the original minimum
			hr := ipComObject.TcSetObjPara(pid := N_PTCID_ForceLimitMin, nData := SIZEOF(stValideMinForce), pData := ADR(stValideMinForce), pgp := 0);
			hr := ipComObject.TcSetObjPara(pid := N_PTCID_ForceLimitMax, nData := SIZEOF(stForceLimitMax), pData := ADR(stForceLimitMax), pgp := 0);
			hr := ipComObject.TcSetObjPara(pid := N_PTCID_ForceLimitMin, nData := SIZEOF(stForceLimitMin), pData := ADR(stForceLimitMin), pgp := 0);
			FW_SafeRelease(ADR(ipComObject));
		END_IF
	
		END_IF
	
		
	20: // Reduce Force to normal			
		fPowerFactor := fMaxForceFactor;
		
		//set force Z, a and b to minimum
		stForceLimitMin := stForceLimitMinAtBeginn;		
		stForceLimitMin.fz := stForceLimitMin.Fz * fPowerFactor;
		stForceLimitMin.Mx := stForceLimitMin.Mx * fPowerFactor;
		stForceLimitMin.My := stForceLimitMin.My * fPowerFactor;
		
		stForceLimitMax := stForceLimitMaxAtBeginn;	
		stForceLimitMax.fz := stForceLimitMax.Fz * fPowerFactor;
		stForceLimitMax.Mx := stForceLimitMax.Mx * fPowerFactor;
		stForceLimitMax.My := stForceLimitMax.My * fPowerFactor;
	    	
		// 13.01.2025 Todo PLC Chash if Min > Max. use objParm insted
		//THIS^.TcIoXPlanarMover.SetForceLimitMax(stForceLimitMax);
		//THIS^.TcIoXPlanarMover.SetForceLimitMin(stForceLimitMin);
		FW_ObjMgr_GetObjectInstance(oid:= THIS^.UtilityTcIoMover.ObjectId, iid:= TC_GLOBAL_IID_LIST.IID_ITComObject, pipUnk:= ADR(ipComObject));
		IF ipComObject <> 0 THEN
			// No minimum can be set if one of the 6 values in the struct is greater than the maximum. Equal is allowed.
			// The minimum is therefore first written to something valid. Followed by Max and the original minimum
			hr := ipComObject.TcSetObjPara(pid := N_PTCID_ForceLimitMin, nData := SIZEOF(stValideMinForce), pData := ADR(stValideMinForce), pgp := 0);
			hr := ipComObject.TcSetObjPara(pid := N_PTCID_ForceLimitMax, nData := SIZEOF(stForceLimitMax), pData := ADR(stForceLimitMax), pgp := 0);
			hr := ipComObject.TcSetObjPara(pid := N_PTCID_ForceLimitMin, nData := SIZEOF(stForceLimitMin), pData := ADR(stForceLimitMin), pgp := 0);
			FW_SafeRelease(ADR(ipComObject));
		END_IF
		
		
		THIS^.UtilityMcMover.SetMaximumPositionLagValue(stLagValuesAtBeginn);
        
		nSeqLiftFromUnknown := 999;
				
	999: // finish seqence feedback
		fbFeedbackLiftFromUnknown.Done := TRUE;
		
	1000..1999:
		//Error
		fbFeedbackLiftFromUnknown.HR := E_FAIL;
END_CASE
END_METHOD

METHOD Halt : HRESULT
VAR_INPUT
END_VAR
THIS^.eActiveCommand 				:= CHALET_NC.E_NcAxisCommands.Halt;
THIS^.fbFeedback.ActiveCommand 		:= TO_STRING(THIS^.eActiveCommand);	
THIS^.fbFeedback.LastCommandAccepted:= TRUE;		
THIS^.fbFeedback.Busy 				:= TRUE;

THIS^.fbMover.Halt(	commandFeedback := THIS^.fbFeedbackHalt, 
					constraint 		:= THIS^.fbDynConstraintContainer 
				   );

Halt := S_OK;
END_METHOD

METHOD MoveA : HRESULT
VAR_INPUT
	fPosition : LREAL;
END_VAR
THIS^.eActiveCommand 				:= CHALET_NC.E_NcAxisCommands.MoveA;
THIS^.fbFeedback.ActiveCommand 		:= TO_STRING(THIS^.eActiveCommand);	
THIS^.fbFeedback.LastCommandAccepted:= TRUE;		
THIS^.fbFeedback.Busy 				:= TRUE;

THIS^.fbMover.MoveA(commandFeedback	:= THIS^.fbFeedbackMoveA, 
					targetPosition	:= fPosition, 
					constraint		:= THIS^.fbDynConstraintContainer
					);

MoveA := S_OK;
END_METHOD

METHOD MoveB : HRESULT
VAR_INPUT
	fPosition : LREAL;
END_VAR
THIS^.eActiveCommand 				:= CHALET_NC.E_NcAxisCommands.MoveB;
THIS^.fbFeedback.ActiveCommand 		:= TO_STRING(THIS^.eActiveCommand);	
THIS^.fbFeedback.LastCommandAccepted:= TRUE;		
THIS^.fbFeedback.Busy 				:= TRUE;

THIS^.fbMover.MoveB(commandFeedback	:= THIS^.fbFeedbackMoveB, 
					targetPosition	:= fPosition, 
					constraint		:= THIS^.fbDynConstraintContainer
					);

MoveB := S_OK;
END_METHOD

METHOD MoveC : HRESULT
VAR_INPUT
	fPosition : LREAL;
	
	(* Addition turns to move in modulo movement (positive or negative). *)
	additionalTurns : UDINT := 0;
	
	(* Direction in which the target is approached. *)
	direction : Tc3_Mc3Definitions.MC_DIRECTION := Tc3_Mc3Definitions.MC_DIRECTION.mcDirectionNonModulo;
END_VAR
VAR
	stMoveCOptions : ST_MoveCOptions;
END_VAR
THIS^.eActiveCommand 				:= CHALET_NC.E_NcAxisCommands.MoveC;
THIS^.fbFeedback.ActiveCommand 		:= TO_STRING(THIS^.eActiveCommand);	
THIS^.fbFeedback.LastCommandAccepted:= TRUE;		
THIS^.fbFeedback.Busy 				:= TRUE;


stMoveCOptions.additionalTurns := additionalTurns;
stMoveCOptions.direction := direction;


THIS^.fbMover.MoveC(commandFeedback	:= THIS^.fbFeedbackMoveC, 
					targetPosition	:= fPosition, 
					constraint		:= THIS^.fbDynConstraintContainer, 
					options			:= stMoveCOptions
					);

MoveC := S_OK;
END_METHOD

METHOD MoveXY : HRESULT
VAR_INPUT
	fPosition_X : LREAL;
	fPosition_Y : LREAL;
END_VAR
VAR
	fbTargetPosition 	: PositionXYC;
	stMoveOptions 		: ST_MoveToPositionOptions;
END_VAR
THIS^.eActiveCommand 				:= CHALET_NC.E_NcAxisCommands.MoveXY;
THIS^.fbFeedback.ActiveCommand 		:= TO_STRING(THIS^.eActiveCommand);	
THIS^.fbFeedback.LastCommandAccepted:= TRUE;		
THIS^.fbFeedback.Busy 				:= TRUE;



fbTargetPosition.SetValuesXY(x := fPosition_X, y := fPosition_Y);

stMoveOptions.useOrientation := TRUE;

THIS^.fbMover.MoveToPosition(	commandFeedback	:= THIS^.fbFeedbackMoveXY, 
								targetPosition	:= fbTargetPosition,
								constraint		:= THIS^.fbDynConstraintContainer, 
								options			:= stMoveOptions);

MoveXY := S_OK;
END_METHOD

METHOD MoveZ : HRESULT
VAR_INPUT
	fPosition : LREAL;
END_VAR
THIS^.eActiveCommand 				:= CHALET_NC.E_NcAxisCommands.MoveZ;
THIS^.fbFeedback.ActiveCommand 		:= TO_STRING(THIS^.eActiveCommand);	
THIS^.fbFeedback.LastCommandAccepted:= TRUE;		
THIS^.fbFeedback.Busy 				:= TRUE;


THIS^.fbMover.MoveZ(commandFeedback	:= THIS^.fbFeedbackMoveZ, 
					targetPosition	:= fPosition, 
					constraint		:= THIS^.fbDynConstraintContainer
					);

MoveZ := S_OK;
END_METHOD

{attribute 'monitoring':='call'}
(* Velocity is zero *)
PROPERTY Standstill : BOOL
GET
Standstill := TRUE;
Standstill := Standstill AND THIS^.PlanarMover.MCTOPLC.SET.SetVelo.x = 0;
Standstill := Standstill AND THIS^.PlanarMover.MCTOPLC.SET.SetVelo.y = 0;
Standstill := Standstill AND THIS^.PlanarMover.MCTOPLC.SET.SetVelo.z = 0;
Standstill := Standstill AND THIS^.PlanarMover.MCTOPLC.SET.SetVelo.a = 0;
Standstill := Standstill AND THIS^.PlanarMover.MCTOPLC.SET.SetVelo.b = 0;
Standstill := Standstill AND THIS^.PlanarMover.MCTOPLC.SET.SetVelo.c = 0;
END_GET
END_PROPERTY

{attribute 'monitoring':='call'}
//The last driving command given had the following value
PROPERTY LastCmdTargetGap : LREAL
GET
LastCmdTargetGap := fLastCmdTargetGap;
END_GET
END_PROPERTY

{attribute 'monitoring':='call'}
//The last driving command given had the following value
PROPERTY LastCmdTargetPosition : LREAL
GET
LastCmdTargetPosition := fLastCmdTargetPosition;
END_GET
END_PROPERTY

{attribute 'monitoring':='call'}
//The last driving command given had the following value
PROPERTY LastCmdTargetTrack: I_XP_Track
GET
LastCmdTargetTrack := ipLastCmdTrack;
END_GET
END_PROPERTY

{attribute 'monitoring':='call'}
//This was the last valid (system enabled) parent station of the mover
PROPERTY LastValidParentStation : I_XP_Station;
GET
VAR_INST

END_VAR
LastValidParentStation := THIS^.ipLastValidParentStation;
END_GET
END_PROPERTY

{attribute 'monitoring':='call'}
//This was the last valid (system enabled) actual  position of the mover
PROPERTY LastValidPositionOnTrack : LREAL
GET
VAR_INST

END_VAR
LastValidPositionOnTrack := THIS^.fLastValidPositionOnTrack;
END_GET
END_PROPERTY

{attribute 'monitoring':='call'}
//This was the last valid (system enabled) actual  position of the mover
PROPERTY LastValidPositionXYZABC : REFERENCE TO MoverVector
GET
VAR_INST

END_VAR
LastValidPositionXYZABC REF= THIS^.stLastValidPositionXYZABC;
END_GET
END_PROPERTY

{attribute 'monitoring':='call'}
//This was the last valid (system enabled) actual  position of the mover
PROPERTY LastValidTrack : I_XP_Track;
GET
VAR_INST

END_VAR
LastValidTrack := THIS^.ipLastValidTrack;
END_GET
END_PROPERTY

{attribute 'monitoring':='call'}
//Distance to the responsible parent station [mm]
PROPERTY DistToParentStation : LREAL
GET
VAR
	fDistToParentStationStartup : LREAL := CHALET_BaseComponents.GVL_Datatypes.cMaxLreal;
	fDistToParentStationReturn : LREAL;
	
	
	ipPath : I_XP_Path;
	bPathFound : BOOL;
	fTempDistToDest : LREAL;
	
	refPosOnTrack : REFERENCE TO MoverVector;
	ipNextWaypoint : I_XP_Station;
	
	fTotalLength : LREAL;
	fDistToBegin : LREAL;
END_VAR
IF THIS^.ParentStation = 0 THEN
	DistToParentStation := CHALET_BaseComponents.GVL_Datatypes.cMaxLreal;
	RETURN;
END_IF

//--- Not on track, line 
IF THIS^.CurrentTrack = 0 THEN
	refPosOnTrack REF= THIS^.ParentStation.PositionOnTrackXYZABC;
	fDistToParentStationReturn := F_DistXYVectors(THIS^.PositionAct,refPosOnTrack);
// ---- ---- ----	


//--- at startup there is no route - parent is station ahead
ELSIF THIS^.fbRouteComplete.IsEmpty THEN
	//check each path behind the parentstation if the mover is on it
	ParentStation.PathsBehinde.ResetIterator();
	WHILE ParentStation.PathsBehinde.HasNextObject() DO
		IF __QUERYINTERFACE(ParentStation.PathsBehinde.GetNextObject(), ipPath) THEN
			//get shortest distance
			fDistToParentStationStartup:= MIN(ipPath.DistanceToDestiantion(ipTrack:= THIS^.CurrentTrack, fPosOnTrack := THIS^.PositionOnTrack), fDistToParentStationStartup);
		END_IF
	END_WHILE
	ParentStation.PathsBehinde.RestoreIterator();	
	fDistToParentStationReturn := fDistToParentStationStartup;
// ---- ---- ----

// ---- Normal route dureing enabled system
ELSE
	THIS^.fbRouteComplete.ResetIterator();
	WHILE THIS^.fbRouteComplete.HasNextObject() DO
		IF __QUERYINTERFACE(THIS^.fbRouteComplete.GetNextObject(), ipPath) THEN
			fTotalLength := fTotalLength + ipPath.Length;
		
			IF NOT bPathFound THEN
				fTempDistToDest := ipPath.DistanceToDestiantion(ipTrack := THIS^.CurrentTrack, fPosOnTrack := THIS^.PositionOnTrack); 
				IF 	fTempDistToDest <> CHALET_BaseComponents.GVL_Datatypes.cMaxLreal THEN
					bPathFound := TRUE;
					fDistToParentStationReturn := fTempDistToDest;
				END_IF
			ELSE 
				fDistToParentStationReturn := fDistToParentStationReturn + ipPath.Length;
			END_IF
		END_IF
	END_WHILE
	THIS^.fbRouteComplete.RestoreIterator();
	// ---- ---- ----
	
	
	//--- If Mover is not on the path, return total length + dist to beginn
	IF NOT bPathFound THEN
		THIS^.fbRouteComplete.ResetIterator();
		IF __QUERYINTERFACE(THIS^.fbRouteComplete.GetNextObject(), ipPath) THEN
			refPosOnTrack REF= ipPath.StationDestination.PositionOnTrackXYZABC;
			fDistToBegin := F_DistXYVectors(THIS^.PositionAct, refPosOnTrack);	
		END_IF
		THIS^.fbRouteComplete.RestoreIterator();
		
		
		fDistToParentStationReturn := fDistToBegin + fTotalLength;
	END_IF
	 // ---- ---- ----

END_IF

DistToParentStation := fDistToParentStationReturn;

//Todo absturz, maximalwert von LREAL überschritten
//redce to 3 decimal places
//DistToParentStation := DINT_TO_LREAL(LREAL_TO_DINT(fDistToParentStationReturn*1000))/1000.0;
END_GET
END_PROPERTY

{attribute 'monitoring':='call'}
//Complete route from last parent to active parent station
PROPERTY RouteComplete : I_CH_List
GET
RouteComplete := THIS^.fbRouteComplete;
END_GET
END_PROPERTY

{attribute 'monitoring':='call'}
//Remaining route to the parent
PROPERTY RouteRemaining: I_CH_List
GET
RouteRemaining := THIS^.fbRouteRemaining;
END_GET
END_PROPERTY

//done segments can be transferred here. these are removed from the remaining route
METHOD RouteSegmentDone : BOOL
VAR_INPUT
	ipPathDone : I_XP_Path;
END_VAR
RouteSegmentDone := THIS^.fbRouteRemaining.RemoveObject(ipPathDone);
END_METHOD

METHOD SetRouteToParent : HRESULT
VAR_INPUT
	ipRoute : I_CH_LIST;
END_VAR
IF ipRoute = 0 THEN
	//Clear on empty input
	THIS^.fbRouteRemaining.Clear();
	THIS^.fbRouteComplete.Clear();
ELSE	
	//set as new route
	THIS^.fbRouteRemaining.Duplicate(ipRoute);
	THIS^.fbRouteComplete.Duplicate(ipRoute);	
END_IF
END_METHOD

{attribute 'monitoring':='call'}
(* Provides the current planar mover setpoint XYZABC [mm/s²] *)
PROPERTY AccelerationSet : REFERENCE TO MoverVector
GET
VAR_INST
	{attribute 'hide'}
	copyOfData :  MoverVector;
END_VAR
//Creat an copy of the struct to view value in targetdbrowser and plc online view
copyOfData := THIS^.fbMover.MCTOPLC.SET.SetAcc;
AccelerationSet REF= copyOfData;
END_GET
END_PROPERTY

{attribute 'monitoring':='call'}
(* C coordinate modulus set in MC3-Planar Mover[°] *)
PROPERTY CAxisModulo : LREAL
GET
VAR
	ipTrackComObject : ITComObject;
	nParaSize : UDINT;
	pParaData : PVOID;
	hr : HRESULT;
	fData : LREAL;
END_VAR
VAR CONSTANT
	N_IDX_OFFSET 	: UDINT := 16#05030107; // Parameter(init) Mover
END_VAR
FW_ObjMgr_GetObjectInstance(oid:= THIS^.OID, iid:= TC_GLOBAL_IID_LIST.IID_ITComObject, pipUnk:= ADR(ipTrackComObject));

IF ipTrackComObject = 0 THEN
	// Error
	RETURN;
END_IF


nParaSize := SIZEOF(fData);	pParaData := ADR(fData);

hr := ipTrackComObject.TcGetObjPara(pid:=N_IDX_OFFSET , nData:= nParaSize, pData:= pParaData, pgp:=0 );
FW_SafeRelease(ADR(ipTrackComObject));


CAxisModulo := TO_LREAL(TO_DINT(fData));
END_GET
END_PROPERTY

{attribute 'monitoring':='call'}
(* Indicates the command mode of an enabled PlanarMover, i.e. how setpoints are currently produced. *)
PROPERTY CommandMode : MC_PLANAR_MOVER_COMMAND_MODE
GET
CommandMode := THIS^.fbMover.MCTOPLC.STD.CommandMode;
END_GET
END_PROPERTY

{attribute 'monitoring':='call'}
//operational and position control active(hovering)
PROPERTY Enabled : BOOL
GET
(* StateDWord bit 20 - operational and position control active *)
Enabled :=  (THIS^.fbMover.MCTOPLC.STD.State = MC_PLANAR_STATE.Enabled) OR
			(THIS^.fbMover.MCTOPLC.STD.State = MC_PLANAR_STATE.Enabling) OR
			(THIS^.fbMover.MCTOPLC.STD.State = MC_PLANAR_STATE.Resetting AND PositionSet.z > 0.0) OR
			(THIS^.fbMover.MCTOPLC.STD.State = MC_PLANAR_STATE.Error AND PositionSet.z > 0.0) OR
			(THIS^.fbMover.MCTOPLC.STD.State = MC_PLANAR_STATE.ErrorPending AND PositionSet.z > 0.0) OR
			(THIS^.fbMover.MCTOPLC.STD.State = MC_PLANAR_STATE.Invalid AND PositionSet.z > 0.0);
END_GET
END_PROPERTY

{attribute 'monitoring':='call'}
(* Retruns lentgh of hypotenuse of the x and y error. (>=0[mm]) *)
PROPERTY LagDistanceXY : LREAL
GET
VAR
	fErrorX, fErrorY : LREAL;
END_VAR
// Set - Act
fErrorX := THIS^.fbMover.MCTOPLC.SET.SetPos.X - THIS^.fbMover.MCTOPLC.ACT.ActPos.X;
fErrorY := THIS^.fbMover.MCTOPLC.SET.SetPos.Y - THIS^.fbMover.MCTOPLC.ACT.ActPos.Y;


//Dist to center. Phytagoras -> c = sqrt( A^2 + B^2)
LagDistanceXY := SQRT(EXPT(fErrorX,2) + EXPT(fErrorY,2));
END_GET
END_PROPERTY

{attribute 'monitoring':='call'}
PROPERTY Mapped : BOOL //Project is mapped to MC (McToPlc and PlcToMc)
GET
VAR
	bMcToPlcNotMapped 	: BOOL;
	bPlcToMcNotMapped 	: BOOL;
END_VAR
//F_GetMappingStatus is not working on IO Data Pointer
	//bPlcToMcNotMapped := F_GetMappingStatus(ADR(THIS^.fbMover.PlcToMc), SIZEOF(THIS^.fbMover.PlcToMc)) <> EPlcMappingStatus.MS_Mapped;
	//bMcToPlcNotMapped := F_GetMappingStatus(ADR(THIS^.fbMover.McToPlc), SIZEOF(THIS^.fbMover.McToPlc)) <> EPlcMappingStatus.MS_Mapped;

	
Mapped := THIS^.fbMover.MCTOPLC.STD.MoverOID <> 0;
END_GET
END_PROPERTY

{attribute 'monitoring':='call'}
PROPERTY Mode : MC_PLANAR_MOVER_COMMAND_MODE
GET
Mode := THIS^.fbMover.MCTOPLC.STD.CommandMode;
END_GET
END_PROPERTY

{attribute 'monitoring':='call'}
(* Height that is used for internal collision checks.[mm] *)
PROPERTY MoverHeight : LREAL
GET
VAR
	ipTrackComObject : ITComObject;
	nParaSize : UDINT;
	pParaData : PVOID;
	hr : HRESULT;
	fData : LREAL;
END_VAR
VAR CONSTANT
	N_IDX_OFFSET 	: UDINT := 16#050300B3; // Parameter(init) Mover
END_VAR
FW_ObjMgr_GetObjectInstance(oid:= THIS^.OID, iid:= TC_GLOBAL_IID_LIST.IID_ITComObject, pipUnk:= ADR(ipTrackComObject));

IF ipTrackComObject = 0 THEN
	// Error
	RETURN;
END_IF


nParaSize := SIZEOF(fData);	pParaData := ADR(fData);

hr := ipTrackComObject.TcGetObjPara(pid:=N_IDX_OFFSET , nData:= nParaSize, pData:= pParaData, pgp:=0 );
FW_SafeRelease(ADR(ipTrackComObject));


MoverHeight := fData;
END_GET
END_PROPERTY

{attribute 'monitoring':='call'}
//Mover could not be detected or was removed from the system
PROPERTY MoverIsNotPresent : BOOL
GET
VAR
	bMoverAtZeroPos, bMoverPositionInvalid, bMoverVeloInvalid : BOOL;
END_VAR
bMoverAtZeroPos		:=  PlanarMover.MCTOPLC.ACT.ActPos.x = 0 AND
						PlanarMover.MCTOPLC.ACT.ActPos.y = 0 AND 
						PlanarMover.MCTOPLC.ACT.ActPos.z = 0 AND 
						PlanarMover.MCTOPLC.ACT.ActPos.a = 0 AND
						PlanarMover.MCTOPLC.ACT.ActPos.b = 0 AND 
						PlanarMover.MCTOPLC.ACT.ActPos.c = 0 AND 
						PlanarMover.MCTOPLC.ACT.PhysicalAreaID = 0;
						
						
bMoverPositionInvalid:=  PlanarMover.MCTOPLC.ACT.ActPos.x >= 1E+302 AND
						PlanarMover.MCTOPLC.ACT.ActPos.y >= 1E+302 AND 
						PlanarMover.MCTOPLC.ACT.ActPos.z >= 1E+302 AND 
						PlanarMover.MCTOPLC.ACT.ActPos.a >= 1E+302 AND
						PlanarMover.MCTOPLC.ACT.ActPos.b >= 1E+302 AND 
						PlanarMover.MCTOPLC.ACT.ActPos.c >= 1E+302;
						
						
bMoverVeloInvalid	:=  PlanarMover.MCTOPLC.ACT.ActVelo.x >= 1E+302 AND
						PlanarMover.MCTOPLC.ACT.ActVelo.y >= 1E+302 AND 
						PlanarMover.MCTOPLC.ACT.ActVelo.z >= 1E+302 AND 
						PlanarMover.MCTOPLC.ACT.ActVelo.a >= 1E+302 AND
						PlanarMover.MCTOPLC.ACT.ActVelo.b >= 1E+302 AND 
						PlanarMover.MCTOPLC.ACT.ActVelo.c >= 1E+302;
						
MoverIsNotPresent := bMoverAtZeroPos OR bMoverPositionInvalid OR bMoverVeloInvalid;
END_GET
END_PROPERTY

{attribute 'monitoring':='call'}
(* Width that is used for internal collision checks.[mm] *)
PROPERTY MoverWidth : LREAL
GET
VAR
	ipTrackComObject : ITComObject;
	nParaSize : UDINT;
	pParaData : PVOID;
	hr : HRESULT;
	fData : LREAL;
END_VAR
VAR CONSTANT
	N_IDX_OFFSET 	: UDINT := 16#050300B2; // Parameter(init) Mover
END_VAR
FW_ObjMgr_GetObjectInstance(oid:= THIS^.OID, iid:= TC_GLOBAL_IID_LIST.IID_ITComObject, pipUnk:= ADR(ipTrackComObject));

IF ipTrackComObject = 0 THEN
	// Error
	RETURN;
END_IF


nParaSize := SIZEOF(fData);	pParaData := ADR(fData);
hr := ipTrackComObject.TcGetObjPara(pid:=N_IDX_OFFSET , nData:= nParaSize, pData:= pParaData, pgp:=0 );
FW_SafeRelease(ADR(ipTrackComObject));

MoverWidth := fData;
END_GET
END_PROPERTY

{attribute 'monitoring':='call'}
(* Contains the information of the Planar Mover passed from MC to PLC. XYZABC [mm] *)
PROPERTY PositionAct : REFERENCE TO MoverVector
GET
VAR_INST
	{attribute 'hide'}
	copyOfActPosition :  MoverVector;
END_VAR
//Creat an copy of the struct to view value in targetdbrowser and plc online view
copyOfActPosition := THIS^.fbMover.MCTOPLC.ACT.ActPos;
PositionAct REF= copyOfActPosition;
END_GET
END_PROPERTY

{attribute 'monitoring':='call'}
(* Provides the current planar mover setpoint XYZABC [mm] *)
PROPERTY PositionSet : REFERENCE TO MoverVector
GET
VAR_INST
	{attribute 'hide'}
	copyOfSetPosition :  MoverVector;
END_VAR
//Creat an copy of the struct to view value in targetdbrowser and plc online view
copyOfSetPosition := THIS^.fbMover.MCTOPLC.SET.SetPos;
PositionSet REF= copyOfSetPosition;
END_GET
END_PROPERTY

{attribute 'monitoring':='call'}
PROPERTY PUBLIC ProductData : I_XP_ProductData
GET
ProductData := ipProductData;
END_GET
SET
// No change. Same interface is set again
IF ipProductData = ProductData THEN
	;//Noting
	
ELSE

	// If allready an interface is linked. Unlink
	IF ipProductData <> 0 THEN
		ipProductData.LinkToMover(0);
		ipProductData := 0;
	END_IF
	
	// Link and store new interface
	IF ProductData <> 0 THEN
		ProductData.LinkToMover(THIS^);
		ipProductData := ProductData;
	END_IF
END_IF
END_SET
END_PROPERTY

{attribute 'monitoring':='call'}
(* Provides the current planar mover act XYZABC [mm/s] *)
PROPERTY VelocityAct : REFERENCE TO MoverVector
GET
VAR_INST
	{attribute 'hide'}
	copyOfData :  MoverVector;
END_VAR
//Creat an copy of the struct to view value in targetdbrowser and plc online view
copyOfData := THIS^.fbMover.MCTOPLC.ACT.ActVelo;
VelocityAct REF= copyOfData;
END_GET
END_PROPERTY

{attribute 'monitoring':='call'}
(* Provides the current planar mover setpoint XYZABC [mm/s] *)
PROPERTY VelocitySet : REFERENCE TO MoverVector
GET
VAR_INST
	{attribute 'hide'}
	copyOfData :  MoverVector;
END_VAR
//Creat an copy of the struct to view value in targetdbrowser and plc online view
copyOfData := THIS^.fbMover.MCTOPLC.SET.SetVelo;
VelocitySet REF= copyOfData;
END_GET
END_PROPERTY

{attribute 'monitoring':='call'}
PROPERTY CurrentTrack : I_XP_Track
GET
VAR
	ipTrackObj : I_CH_Object;
	ipTrack : I_XP_Track;
END_VAR
IF ipXpSystem <> 0 THEN
	ipTrackObj := ipXpSystem.Tracks.FindOID(THIS^.PlanarMover.MCTOPLC.SETONTRACK.TrackOID);
	ToXpTrack(ipTrackObj,ipTrack);
END_IF

CurrentTrack := ipTrack;
END_GET
END_PROPERTY

METHOD DistToTrack : LREAL
VAR_INPUT
	iTrack : I_XP_Track;
END_VAR
VAR
	fPositionOnTrack : LREAL;
	trackPosition, moverPosition : PositionXYC;
END_VAR
moverPosition.x := PositionSet.x;
moverPosition.y := PositionSet.y;
moverPosition.c := PositionSet.c;

//Get Pos on track in mm
fPositionOnTrack := iTrack.PlanarTrack.GetArcLengthClosestTo(geometry:=moverPosition);

//Convert pos on track in XY
iTrack.PlanarTrack.GetPositionAt(arcLength := fPositionOnTrack, position:=trackPosition);

//Get distance to mover
DistToTrack := SQRT(EXPT((trackPosition.x - moverPosition.x),2)+EXPT((trackPosition.y - moverPosition.y),2));
END_METHOD

METHOD JoinTrack : HRESULT
VAR_INPUT
	iTrack : I_XP_Track;
END_VAR
VAR
	joinTrackOptions : ST_JoinTrackOptions;
END_VAR
IF iTrack <> 0 THEN
	THIS^.eActiveCommand 				:= CHALET_NC.E_NcAxisCommands.JoinTrack;
	THIS^.fbFeedback.ActiveCommand 		:= TO_STRING(THIS^.eActiveCommand);	
	THIS^.fbFeedback.LastCommandAccepted:= TRUE;		
	THIS^.fbFeedback.Busy 				:= TRUE;

	
	(* ADS Error 33164 or 33154: Position out of modulo range or Software position limit violation. Position must be larger or equal to zero and less or equal to the modulus when using modulo positioning. 
		When using modulo positioning, the target position is interpreted in consideration of the AdditionalTurns variable at the Options input.

		If the above error occurs, then the mover wants to rotate on the track when joining because ‘useOrientation = TRUE’ is set. 
		Better do not to set this to false, because CA then requires a much greater distance to the neighbouring mover.
		It is better to check the set C-axis modules in the MC3 PlanarMover if 90, 180 or 360°.
	*)
	joinTrackOptions.useOrientation 	:= TRUE;

	
	THIS^.fbMover.JoinTrack(commandFeedback	:= THIS^.fbFeedbackJoinTrack, 
								targetTrack	:= iTrack.PlanarTrack, 
								constraint	:= THIS^.fbDynConstraintContainer,
								options		:= joinTrackOptions);								
	JoinTrack := S_OK;
ELSE
	JoinTrack := S_FALSE;
	THIS^.fbFeedback.LastCommandAccepted:= FALSE;	
END_IF
END_METHOD

METHOD MoveOnTrack : HRESULT
VAR_INPUT
	ipTrack : I_XP_Track;
	fPosition : LREAL;
	fGap : LREAL;
END_VAR

VAR
	moveOptions: ST_MoveOnTrackOptions;
	//fMoverDiagonal : LREAL;
END_VAR
moveOptions.direction := Tc3_Mc3Definitions.MC_DIRECTION.mcDirectionPositive;
moveOptions.additionalTurns := 0;
moveOptions.gap := XPlanarParameterlist.N_GAP_MODE_ON_TRACK; 

//Use fix gap if requested gap is to small
moveOptions.gap := MAX(fGap, XPlanarParameterlist.F_MOVER_MINIMUM_GAP_ON_TRACK);
moveOptions.dynamicMode := XPlanarParameterlist.N_SELECT_MODE_HOW_DYNAMIC_IS_PLANED_ON_TRACK;

IF ipTrack <> 0 THEN
	THIS^.eActiveCommand 				:= CHALET_NC.E_NcAxisCommands.MoveOnTrack;
	THIS^.fbFeedback.ActiveCommand 		:= TO_STRING(THIS^.eActiveCommand);	
	THIS^.fbFeedback.LastCommandAccepted:= TRUE;		
	THIS^.fbFeedback.Busy 				:= TRUE;

	THIS^.fbMover.MoveOnTrack(
		commandFeedback			:= THIS^.fbFeedbackMoveOnTrack,
		targetTrack				:= ipTrack.PlanarTrack, 
		targetPositionOnTrack	:= fPosition, 
		constraint				:= THIS^.fbDynConstraintPath, 
		options					:= moveOptions);
	
	//Store the values
	fLastCmdTargetPosition 	:= fPosition; //the last commanded target position [mm]
	fLastCmdTargetGap 		:= moveOptions.gap; //the last commanded target gap
	ipLastCmdTrack		 	:= ipTrack; //the last commanded target track	
	
	
	MoveOnTrack := S_OK;
ELSE
	MoveOnTrack := S_FALSE;
	THIS^.fbFeedback.LastCommandAccepted:= FALSE;	
END_IF
END_METHOD

METHOD MoveOnTrack_ShortestWay : HRESULT
VAR_INPUT
	ipTrack : I_XP_Track;
	fPosition : LREAL;
	fGap : LREAL;
END_VAR

VAR
	moveOptions: ST_MoveOnTrackOptions;
	//fMoverDiagonal : LREAL;
END_VAR
moveOptions.direction := Tc3_Mc3Definitions.MC_DIRECTION.mcDirectionShortestWay;
moveOptions.additionalTurns := 0;
moveOptions.gap := XPlanarParameterlist.N_GAP_MODE_ON_TRACK; 

//Use fix gap if requested gap is to small
moveOptions.gap := MAX(fGap, XPlanarParameterlist.F_MOVER_MINIMUM_GAP_ON_TRACK);
moveOptions.dynamicMode := XPlanarParameterlist.N_SELECT_MODE_HOW_DYNAMIC_IS_PLANED_ON_TRACK;

IF ipTrack <> 0 THEN
	THIS^.eActiveCommand 				:= CHALET_NC.E_NcAxisCommands.MoveOnTrack;		
	THIS^.fbFeedback.ActiveCommand 		:= TO_STRING(THIS^.eActiveCommand);	
	THIS^.fbFeedback.LastCommandAccepted:= TRUE;		
	THIS^.fbFeedback.Busy 				:= TRUE;
	
	THIS^.fbMover.MoveOnTrack(
		commandFeedback			:= THIS^.fbFeedbackMoveOnTrack,
		targetTrack				:= ipTrack.PlanarTrack, 
		targetPositionOnTrack	:= fPosition, 
		constraint				:= THIS^.fbDynConstraintPath, 
		options					:= moveOptions);
				
	fLastCmdTargetPosition 	:= fPosition; //the last commanded target position [mm]
	fLastCmdTargetGap 		:= moveOptions.gap; //the last commanded target gap
	ipLastCmdTrack		 	:= ipTrack; //the last commanded target track	
		
	MoveOnTrack_ShortestWay := S_OK;
ELSE
	MoveOnTrack_ShortestWay := S_FALSE;
	THIS^.fbFeedback.LastCommandAccepted:= FALSE;	
END_IF
END_METHOD

METHOD MoveOnTrackToStation : HRESULT
VAR_INPUT
	ipStation : I_XP_Station;
	fGap : LREAL;
END_VAR
IF ipStation <> 0 AND_THEN ipStation.AccocietedTrack <> 0 THEN

	MoveOnTrackToStation := MoveOnTrack(ipTrack:= ipStation.AccocietedTrack, 
										fPosition:= ipStation.PositionOnTrack, 
										fGap:= fGap);
ELSE
	MoveOnTrackToStation := E_FAIL;
	THIS^.fbFeedback.LastCommandAccepted:= FALSE;	
END_IF
END_METHOD

{attribute 'monitoring':='call'}
PROPERTY ParentStation : I_XP_Station
GET
ParentStation := ipParentStation;
END_GET
SET
THIS^.ipParentStation := ParentStation;

IF ParentStation <> 0 THEN
	THIS^.ipLastValidParentStation := ParentStation;
END_IF
END_SET
END_PROPERTY

{attribute 'monitoring':='call'}
PROPERTY PositionOnTrack : LREAL
GET
VAR_INST
	{attribute 'hide'}	
	fPosOnTrack : LREAL;
END_VAR
fPosOnTrack := THIS^.fbMover.MCTOPLC.SETONTRACK.SetPos;
PositionOnTrack := fPosOnTrack;
END_GET
END_PROPERTY

{attribute 'monitoring':='call'}
PROPERTY TargetStation : STRING
GET
TargetStation := THIS^.sTargetStation;
END_GET
SET
THIS^.sTargetStation := TargetStation;
END_SET
END_PROPERTY

{attribute 'monitoring':='call'}
PROPERTY UtilityMcMover : Tc3_XPlanarUtility.I_McPlanarMover
GET
UtilityMcMover :=  THIS^.ipMcMover;
END_GET
END_PROPERTY

{attribute 'monitoring':='call'}
PROPERTY UtilityTcIoMover : Tc3_XPlanarUtility.I_TcIoXPlanarMover
GET
VAR
;
END_VAR
UtilityTcIoMover := THIS^.ipTcIoMover;
END_GET
END_PROPERTY

METHOD FB_init : BOOL
VAR_INPUT
	bInitRetains : BOOL; // if TRUE, the retain variables are initialized (warm start / cold start)
	bInCopyCode : BOOL;  // if TRUE, the instance afterwards gets moved into the copy code (online change)
	
	
	ipSystem : I_CH_Object;
END_VAR
//Do the following code once during start up and not during onlinechange
IF NOT bInCopyCode THEN 
	
	
	(* Register to the Xplanar System
	   1. Test if the interface exists
	   2. Test if the object implements a "System for Mover" interface 
	*)
	IF ipSystem <> 0 AND_THEN __QUERYINTERFACE(ipSystem,THIS^.ipXpSystem) THEN
		THIS^.ipXpSystem.RegisterMover(THIS^);
	END_IF

	
	
	THIS^.fbFeedback.ActiveCommand 		:= TO_STRING(THIS^.eActiveCommand);	
	
	
END_IF
END_METHOD

{attribute 'monitoring':='call'}
PROPERTY Feedback : I_XP_Feedback
GET
Feedback := THIS^.fbFeedback;
END_GET
END_PROPERTY

METHOD Initialize : HRESULT
VAR
	bWaitForAxisInit : BOOL;
	hrExtAxis : HRESULT;
	stVarInfo : __SYSTEM.VAR_INFO;
	
	nIdxXpu : UDINT;
	nIdxMover : UDINT;
	ipTcIoXpu : I_TcIoXPlanarProcessingUnit;	
	//nMoverOID : OTCID;
	nOidHardwareMover : OTCID;
	hr : HRESULT;
	ipComObject : ITComObject;
	nParaSize : UDINT;
	pParaData : PVOID;
END_VAR
VAR CONSTANT
	N_IDX_HARDWARE_MOVER_OID 	: UDINT := 16#0503012D; // Parameter(online) "Hardware mover OTCID"
END_VAR

VAR_INST
	//This error cannot be reset. Requires a reset cold
	{attribute 'hide'}	
	fbInitError : FB_TcAlarm;
END_VAR
// Check if link to MC-Mover is mapped
IF NOT THIS^.Mapped THEN
	IF NOT fbInitError.bRaised THEN 
		//This error cannot be reset. Requires a reset cold
		fbInitError.CreateEx(stEventEntry:=TC_EVENTS.CHALET_Base_Events.VariableLinkMissing, ipSourceInfo := THIS^.fbSourceInfo, bWithConfirmation := FALSE);
		stVarInfo := __VARINFO(fbMover);
		fbInitError.ipArguments.AddString(stVarInfo.Symbol);
		fbInitError.Raise(0);
	END_IF
	Initialize := E_FAIL;
	RETURN;
END_IF


	
IF NOT bInitDone THEN
	//Get MC-Mover interface to utiliy lib
	FOR nIdxMover := 1 TO ipXpSystem.Enviroment.UtilityEnvirement.P_MoverCount DO
		IF ipXpSystem.Enviroment.UtilityEnvirement.P_MoverOids[nIdxMover] = THIS^.fbMover.MCTOPLC.STD.MoverOID THEN
			THIS^.ipMcMover := ipXpSystem.Enviroment.UtilityEnvirement.McMover(nIdxMover);
			EXIT;
		END_IF
	END_FOR

	
	//get OID of to MC-Mover mapped TcIoMover
	hr := FW_ObjMgr_GetObjectInstance(oid:= THIS^.fbMover.MCTOPLC.STD.MoverOID, iid:= TC_GLOBAL_IID_LIST.IID_ITComObject, pipUnk:= ADR(ipComObject));
	IF ipComObject <> 0 THEN
		//Get ADR and SIZE
		nParaSize := SIZEOF(nOidHardwareMover);	pParaData := ADR(nOidHardwareMover);
		hr := ipComObject.TcGetObjPara(pid:=N_IDX_HARDWARE_MOVER_OID , nData:= nParaSize, pData:= pParaData, pgp:=0 );
		FW_SafeRelease(ADR(ipComObject));
		
		IF nOidHardwareMover = 0 THEN
			//TODO Errormessage. MC is not mapped to TcIO
			RETURN;
		END_IF
	
		//Search interface for this OID
		FOR nIdxXpu := 1 TO ipXpSystem.Enviroment.UtilityEnvirement.P_XpuCount DO
			ipTcIoXpu := ipXpSystem.Enviroment.UtilityEnvirement.TcIoXpu(nIdxXpu);
			
			IF ipTcIoXpu <> 0 THEN
				//Get TcIo-Mover interface to utiliy lib
				FOR nIdxMover := 1 TO Param_TcIoXPlanarEnvironment.MaxXPlanarMoversPerXpu DO
					IF ipTcIoXpu.P_MoverOids[nIdxMover] = nOidHardwareMover THEN
						THIS^.ipTcIoMover := ipTcIoXpu.TcIoMover(nIdxMover);
						EXIT;
					END_IF
				END_FOR
			END_IF
		END_FOR	
	END_IF
	
	IF THIS^.ipTcIoMover = 0 OR THIS^.ipMcMover = 0 THEN
		//TODO Errormessage. Utility interface not found
		RETURN;
	END_IF
	

	//Set all move dynamic constraint to the axis default value.
	THIS^.SetDynConstraint_X(MC_DEFAULT,MC_DEFAULT,MC_DEFAULT,MC_DEFAULT);
	THIS^.SetDynConstraint_Y(MC_DEFAULT,MC_DEFAULT,MC_DEFAULT,MC_DEFAULT);	
	THIS^.SetDynConstraint_Z(MC_DEFAULT,MC_DEFAULT,MC_DEFAULT,MC_DEFAULT);	
	THIS^.SetDynConstraint_A(MC_DEFAULT,MC_DEFAULT,MC_DEFAULT,MC_DEFAULT);	
	THIS^.SetDynConstraint_B(MC_DEFAULT,MC_DEFAULT,MC_DEFAULT,MC_DEFAULT);
	THIS^.SetDynConstraint_C(MC_DEFAULT,MC_DEFAULT,MC_DEFAULT,MC_DEFAULT);
	THIS^.SetDynConstraint_Path(MC_DEFAULT,MC_DEFAULT,MC_DEFAULT,MC_DEFAULT);

	//Call Init of Setpointaxis only, if mapped
	IF AxisSetpointX.Mapped THEN hrExtAxis := GetMostSignificant(hrExtAxis, AxisSetpointX.Initialize());END_IF
	IF AxisSetpointY.Mapped THEN hrExtAxis := GetMostSignificant(hrExtAxis, AxisSetpointY.Initialize());END_IF
	IF AxisSetpointZ.Mapped THEN hrExtAxis := GetMostSignificant(hrExtAxis, AxisSetpointZ.Initialize());END_IF
	IF AxisSetpointA.Mapped THEN hrExtAxis := GetMostSignificant(hrExtAxis, AxisSetpointA.Initialize());END_IF
	IF AxisSetpointB.Mapped THEN hrExtAxis := GetMostSignificant(hrExtAxis, AxisSetpointB.Initialize());END_IF
	IF AxisSetpointC.Mapped THEN hrExtAxis := GetMostSignificant(hrExtAxis, AxisSetpointC.Initialize());END_IF	
	
	bInitDone := (hrExtAxis = S_OK);	
	
	
	//Pending
	Initialize := S_PENDING;;	
ELSE	
	//Done
	Initialize := S_OK;	
END_IF


THIS^.eActiveCommand 				:= CHALET_NC.E_NcAxisCommands.Initialize;
THIS^.fbFeedback.ActiveCommand 		:= TO_STRING(THIS^.eActiveCommand);	
THIS^.fbFeedback.LastCommandAccepted:= TRUE;	
//Set done or keep in busy state	
THIS^.fbFeedback.HR := Initialize;
END_METHOD

{attribute 'monitoring':='call'}
//Unique object ID
PROPERTY OID : OTCID
GET
OID := THIS^.fbMover.MCTOPLC.STD.MoverOID;
END_GET
END_PROPERTY

{attribute 'monitoring':='call'}
PROPERTY PlanarMover : REFERENCE TO MC_PlanarMover
GET
PlanarMover ref= THIS^.fbMover;
END_GET
END_PROPERTY

(* Time-critical information is processed here, which can then be polled via the property every cycle. 
The update method is usually at the end of the program and then it is already 'outdated'. *)
METHOD PRIVATE Prepare : HRESULT
VAR

END_VAR
VAR_INST
	{attribute 'hide'}
	nLastUpdatedCycleCount : UDINT;
END_VAR
//Check if this Cycle the dates are allready prepared
IF nLastUpdatedCycleCount <> TwinCAT_SystemInfoVarList._TaskInfo[THIS^.nTaskIndex].CycleCount THEN
	nLastUpdatedCycleCount := TwinCAT_SystemInfoVarList._TaskInfo[THIS^.nTaskIndex].CycleCount;

	//Stor last valide position im system is enabled
	IF ipXpSystem.Enabled THEN
		THIS^.stLastValidPositionXYZABC := THIS^.PositionSet;
		THIS^.fLastValidPositionOnTrack := THIS^.PositionOnTrack;
		THIS^.ipLastValidTrack := THIS^.CurrentTrack;
	END_IF

END_IF
END_METHOD

{attribute 'monitoring':='call'}
//Interface to CHALET system to which this object belongs
PROPERTY System : I_XP_System_PLC
GET
//get I_x_System_PLC interface from I_x_System_Registration
__QUERYINTERFACE(THIS^.ipXpSystem, System);
END_GET
END_PROPERTY

METHOD PUBLIC Update : HRESULT
VAR
	ipObject : I_CH_Object;
END_VAR

VAR_INST
	{attribute 'hide'}
	fbCmdNotPossibleCollision : FB_TcAlarm;
	{attribute 'hide'}
	nFeedbackOidOld : UDINT;
	{attribute 'hide'}	
	nOldNcErrorCode 		: UDINT;
	{attribute 'hide'}	
	fbAlarmNcErrorCode		: FB_TcAlarm;
END_VAR
THIS^.Prepare();//Prepare time-critical information, if not already done

THIS^.UpdateExternalSetpoint();
THIS^.UpdateUnknownLevel();

// ********************** Set feedback depending on active command *******************************
CASE THIS^.eActiveCommand OF
	E_NcAxisCommands.None: 
		//Display if a Mover Error is active during no command is active
		IF THIS^.fbMover.Error AND NOT fbFeedback.Error THEN 
			IF THIS^.fbMover.ErrorId <> 1810(*ignore ADSERR_DEVICE_INVALIDSTATE*) THEN
				fbFeedback.ErrorId 			:= THIS^.fbMover.ErrorID;
				fbFeedback.ActiveCommand 	:= TO_STRING(E_NcAxisCommands.None);	
				fbFeedback.ClearObjectInfo();
			END_IF
		END_IF

	E_NcAxisCommands.Initialize:
		fbFeedback.Busy 			:= NOT THIS^.bInitDone;
		fbFeedback.Done 			:= THIS^.bInitDone;
		fbFeedback.ErrorId 			:= 0;
		fbFeedback.ClearObjectInfo();
		                        	
	E_NcAxisCommands.MoveA:     	
		fbFeedback.Busy 			:= fbFeedbackMoveA.Busy;
		fbFeedback.Done 			:= fbFeedbackMoveA.Done;
		fbFeedback.ErrorId 			:= fbFeedbackMoveA.ErrorID;
        fbFeedback.ObjectInfo		:= fbFeedbackMoveA.objectInfo;
                                	
	E_NcAxisCommands.MoveB:     	
		fbFeedback.Busy 			:= fbFeedbackMoveB.Busy;
		fbFeedback.Done 			:= fbFeedbackMoveB.Done;
		fbFeedback.ErrorId 			:= fbFeedbackMoveB.ErrorID;
        fbFeedback.ObjectInfo		:= fbFeedbackMoveB.objectInfo;
                                	
	E_NcAxisCommands.MoveC:     	
		fbFeedback.Busy 			:= fbFeedbackMoveC.Busy;
		fbFeedback.Done 			:= fbFeedbackMoveC.Done;
		fbFeedback.ErrorId 			:= fbFeedbackMoveC.ErrorID;
        fbFeedback.ObjectInfo		:= fbFeedbackMoveC.objectInfo;
                                	
	E_NcAxisCommands.MoveXY:    	
		fbFeedback.Busy 			:= fbFeedbackMoveXY.Busy;
		fbFeedback.Done 			:= fbFeedbackMoveXY.Done;
		fbFeedback.ErrorId 			:= fbFeedbackMoveXY.ErrorID;
        fbFeedback.ObjectInfo		:= fbFeedbackMoveXY.objectInfo;
                                	
	E_NcAxisCommands.MoveZ:     	
		fbFeedback.Busy 			:= fbFeedbackMoveZ.Busy;
		fbFeedback.Done 			:= fbFeedbackMoveZ.Done;
		fbFeedback.ErrorId 			:= fbFeedbackMoveZ.ErrorID;
        fbFeedback.ObjectInfo		:= fbFeedbackMoveZ.objectInfo;
                                	
	E_NcAxisCommands.Enable:    	
		fbFeedback.Busy 			:= fbFeedbackEnable.Busy;
		fbFeedback.Done 			:= fbFeedbackEnable.Done;
		fbFeedback.ErrorId 			:= fbFeedbackEnable.ErrorID;
        fbFeedback.ObjectInfo		:= fbFeedbackEnable.objectInfo;
                                	
	E_NcAxisCommands.Disable:   	
		fbFeedback.Busy 			:= fbFeedbackDisable.Busy;
		fbFeedback.Done 			:= fbFeedbackDisable.Done;
		fbFeedback.ErrorId 			:= fbFeedbackDisable.ErrorID;
        fbFeedback.ObjectInfo		:= fbFeedbackDisable.objectInfo;
                                	
	E_NcAxisCommands.Reset:     	
		fbFeedback.Busy 			:= fbFeedbackReset.Busy;
		fbFeedback.Done 			:= fbFeedbackReset.Done;
		fbFeedback.ErrorId 			:= fbFeedbackReset.ErrorID;
        fbFeedback.ObjectInfo		:= fbFeedbackReset.objectInfo;
                                	
	E_NcAxisCommands.Halt:      	
		fbFeedback.Busy 			:= fbFeedbackHalt.Busy;
		fbFeedback.Done 			:= fbFeedbackHalt.Done;
		fbFeedback.ErrorId 			:= fbFeedbackHalt.ErrorID;
        fbFeedback.ObjectInfo		:= fbFeedbackHalt.objectInfo;

	E_NcAxisCommands.AddToGroupe:
		fbFeedback.Busy 			:= fbFeedbackAddToGrp.Busy;
		fbFeedback.Done 			:= fbFeedbackAddToGrp.Done;
		fbFeedback.ErrorId 			:= fbFeedbackAddToGrp.ErrorID;
        fbFeedback.ObjectInfo		:= fbFeedbackAddToGrp.objectInfo;

	E_NcAxisCommands.RemoveFromGroupe:
		fbFeedback.Busy 			:= fbFeedbackRmvFromGrp.Busy;
		fbFeedback.Done 			:= fbFeedbackRmvFromGrp.Done;
		fbFeedback.ErrorId 			:= fbFeedbackRmvFromGrp.ErrorID;
        fbFeedback.ObjectInfo		:= fbFeedbackRmvFromGrp.objectInfo;
		
	E_NcAxisCommands.JoinTrack:
		fbFeedback.Busy 			:= fbFeedbackJoinTrack.Busy;
		fbFeedback.Done 			:= fbFeedbackJoinTrack.Done;
		fbFeedback.ErrorId 			:= fbFeedbackJoinTrack.ErrorID;
        fbFeedback.ObjectInfo		:= fbFeedbackJoinTrack.objectInfo;
		
	E_NcAxisCommands.MoveOnTrack:
		fbFeedback.Busy 			:= fbFeedbackMoveOnTrack.Busy;
		fbFeedback.Done 			:= fbFeedbackMoveOnTrack.Done;
		fbFeedback.ErrorId 			:= fbFeedbackMoveOnTrack.ErrorID;
        fbFeedback.ObjectInfo		:= fbFeedbackMoveOnTrack.objectInfo;
		
			
	E_NcAxisCommands.StartExternalSetpoint:
		;// in Subroutine "UpdateExternalSetpoint"
	
	E_NcAxisCommands.StopExternalSetpoint:
		;// in Subroutine "UpdateExternalSetpoint"		
			
	E_NcAxisCommands.LiftFromUnknownLevel:
		fbFeedback.Busy 			:= fbFeedbackLiftFromUnknown.Busy;
		fbFeedback.Done 			:= fbFeedbackLiftFromUnknown.Done;
		fbFeedback.ErrorId 			:= fbFeedbackLiftFromUnknown.ErrorID;
        fbFeedback.ClearObjectInfo();
	
	E_NcAxisCommands.LowerToUnknownLevel:
		fbFeedback.Busy 			:= fbFeedbackLowerToUnknown.Busy;
		fbFeedback.Done 			:= fbFeedbackLowerToUnknown.Done;
		fbFeedback.ErrorId 			:= fbFeedbackLowerToUnknown.ErrorID;
        fbFeedback.ClearObjectInfo();
		
	ELSE//External command in subclass
		;
END_CASE


// **********************  Stop to execute commands on .done or .error ***************************
IF fbFeedback.Done OR THIS^.fbFeedback.Error THEN
	eActiveCommand 				:= E_NcAxisCommands.None;
END_IF


// **********************  Get interface to Feedback.ObjectInfo ***************************
IF Feedback.ObjectInfoEx.Id <> 0 AND Feedback.ObjectInfoEx.Id <> nFeedbackOidOld THEN
	CASE Feedback.ObjectInfo.ObjectType OF
		EPlanarObjectType.Mover:
			Feedback.ObjectInfoEx.ipObject := THIS^.ipXPSystem.MoversPresent.FindOID(Feedback.ObjectInfo.Id);
			
		EPlanarObjectType.Track:
				Feedback.ObjectInfoEx.ipObject := THIS^.ipXPSystem.Tracks.FindOID(Feedback.ObjectInfo.Id);
		
		EPlanarObjectType.Environment:
				Feedback.ObjectInfoEx.ipObject := THIS^.ipXPSystem.Enviroment;
				
		ELSE 
			Feedback.ObjectInfoEx.ipObject := 0;
	END_CASE
END_IF
nFeedbackOidOld := Feedback.ObjectInfo.Id;



// **********************  Write NC-Error(Mover.MCTOPLC.ErrorCode) in TC3 Eventlogger ***************************
IF (THIS^.fbMover.MCTOPLC.STD.ErrorCode = 0 AND fbAlarmNcErrorCode.bRaised) THEN
	//No error - Reset	
	fbAlarmNcErrorCode.Clear(0,0);
	
ELSIF (THIS^.fbMover.MCTOPLC.STD.ErrorCode = 0) THEN
	; //Nothing
	
ELSIF (nOldNcErrorCode <> THIS^.fbMover.MCTOPLC.STD.ErrorCode) THEN
	//New Error - Reset, Create and Raise
	fbAlarmNcErrorCode.Clear(0,0);
	fbAlarmNcErrorCode.Create(	eventClass		:= TC_EVENT_CLASSES.Tc3_NcErrorCodes, 
								nEventId		:= (TO_DWORD(THIS^.fbMover.MCTOPLC.STD.ErrorCode) AND 16#FFFF), //Cut HRESULT to 4 digit error code
								eSeverity		:= TcEventSeverity.Error, 
								ipSourceInfo 	:= THIS^.fbSourceInfo, 
								bWithConfirmation := FALSE);
	fbAlarmNcErrorCode.ipArguments.Clear();
	fbAlarmNcErrorCode.Raise(0);
ELSE
	//Alarm is already active
	;
END_IF
nOldNcErrorCode := THIS^.fbMover.MCTOPLC.STD.ErrorCode;



// **********************  Raise alarm on collision error ***************************
ipObject := THIS^.fbFeedback.ObjectInfoEx.ipObject;
IF THIS^.fbFeedback.Error AND (ipObject <> 0) AND NOT fbCmdNotPossibleCollision.bRaised THEN
	fbCmdNotPossibleCollision.CreateEx(stEventEntry := TC_EVENTS.CHALET_XPlanar_Events.CommandNotPossibleCollision, bWithConfirmation := FALSE, ipSourceInfo := THIS^.fbSourceInfo);
	//Command "{1}" not possible. Possible collision with "{2}"
	fbCmdNotPossibleCollision.ipArguments.AddStringByValue(THIS^.fbFeedback.ActiveCommand).AddStringByValue(ipObject.LUID);
	fbCmdNotPossibleCollision.Raise(0);
ELSIF NOT THIS^.fbFeedback.Error OR ipObject = 0 THEN
	fbCmdNotPossibleCollision.Clear(0,0);	
END_IF




//Update xplanar object
THIS^.fbMover.Update();



//Update feedback object
fbFeedbackMoveA.Update(); 
fbFeedbackMoveB.Update(); 
fbFeedbackMoveC.Update(); 
fbFeedbackMoveXY.Update(); 
fbFeedbackMoveZ.Update(); 
fbFeedbackEnable.Update(); 
fbFeedbackDisable.Update(); 
fbFeedbackReset.Update(); 
fbFeedbackAddToGrp.Update(); 
fbFeedbackRmvFromGrp.Update(); 
fbFeedbackHalt.Update(); 
fbFeedbackJoinTrack.Update(); 
fbFeedbackMoveOnTrack.Update();
END_METHOD

END_FUNCTION_BLOCK

// FUNCTIONs/F_Vector_Subtraction
FUNCTION F_Vector_Subtraction : MoverVector //difference.x = minuend.x - subtrahend.x
VAR_INPUT
	minuend : REFERENCE TO MoverVector;
	subtrahend : REFERENCE TO MoverVector;
END_VAR
VAR
	
END_VAR

IF NOT __ISVALIDREF(minuend) OR NOT __ISVALIDREF(subtrahend) THEN
	//Error
	RETURN;
END_IF

F_Vector_Subtraction.x	:= minuend.x	- subtrahend.x;
F_Vector_Subtraction.y	:= minuend.y	- subtrahend.y;
F_Vector_Subtraction.z	:= minuend.z	- subtrahend.z;
F_Vector_Subtraction.a	:= minuend.a	- subtrahend.a;
F_Vector_Subtraction.b	:= minuend.b	- subtrahend.b;
F_Vector_Subtraction.c	:= minuend.c	- subtrahend.c;

END_FUNCTION

// FUNCTIONs/F_Vector_Multiplication
FUNCTION F_Vector_Multiplication : MoverVector //product.x = factor1.x * factor2.x
VAR_INPUT
	factor1 : REFERENCE TO MoverVector;
	factor2 : REFERENCE TO MoverVector;
END_VAR
VAR
	
END_VAR

IF NOT __ISVALIDREF(factor1) OR NOT __ISVALIDREF(factor2) THEN
	//Error
	RETURN;
END_IF

F_Vector_Multiplication.x	:= factor1.x	* factor2.x;
F_Vector_Multiplication.y	:= factor1.y	* factor2.y;
F_Vector_Multiplication.z	:= factor1.z	* factor2.z;
F_Vector_Multiplication.a	:= factor1.a	* factor2.a;
F_Vector_Multiplication.b	:= factor1.b	* factor2.b;
F_Vector_Multiplication.c	:= factor1.c	* factor2.c;

END_FUNCTION

// FUNCTIONs/F_Vector_Addition
FUNCTION F_Vector_Addition : MoverVector //sum = summand1 + summand2
VAR_INPUT
	summand1 : REFERENCE TO MoverVector;
	summand2 : REFERENCE TO MoverVector;
END_VAR
VAR
	
END_VAR

IF NOT __ISVALIDREF(summand1) OR NOT __ISVALIDREF(summand2) THEN
	//Error
	RETURN;
END_IF

F_Vector_Addition.x	:= summand1.x	+ summand2.x;
F_Vector_Addition.y	:= summand1.y	+ summand2.y;
F_Vector_Addition.z	:= summand1.z	+ summand2.z;
F_Vector_Addition.a	:= summand1.a	+ summand2.a;
F_Vector_Addition.b	:= summand1.b	+ summand2.b;
F_Vector_Addition.c	:= summand1.c	+ summand2.c;

END_FUNCTION

// COMPONENTs/Optional/Casting/ToXpTrack
FUNCTION ToXpTrack : BOOL
VAR_INPUT
	iChObject : I_CH_OBJECT;
	iXpTrack : REFERENCE TO I_XP_Track;
END_VAR

VAR
	iTmp : I_XP_Track;
END_VAR

(* 
   1. Test if the interface exists
   2. Test if the object implements a "Object" interface 
   3. Write reference to interface in parameter
   4. Returne TRUE if succesfull
*)
IF iChObject <> 0 AND_THEN __QUERYINTERFACE(iChObject,iTmp) THEN
	iXpTrack := iTmp;
	ToXpTrack := TRUE;
END_IF

END_FUNCTION

// COMPONENTs/Optional/Casting/ToXpMover
FUNCTION ToXpMover : BOOL
VAR_INPUT
	iChObject : I_CH_OBJECT;
	iXpMover : Reference to I_XP_Mover;
END_VAR

VAR
	iTmp : I_XP_Mover;
END_VAR

(* 
   1. Test if the interface exists
   2. Test if the object implements a "Object" interface 
   3. Write reference to interface in parameter
   4. Returne TRUE if succesfull
*)
IF iChObject <> 0 AND_THEN __QUERYINTERFACE(iChObject,iTmp) THEN
	iXpMover := iTmp;
	ToXpMover := TRUE;
END_IF

END_FUNCTION

// COMPONENTs/Optional/Casting/ToXpStation
FUNCTION ToXpStation : BOOL
VAR_INPUT
	iChObject : I_CH_OBJECT;
	iXpStation : REFERENCE TO I_XP_Station;
END_VAR

VAR
	iTmp : I_XP_Station;
END_VAR

(* Register the Station
   1. Test if the interface exists
   2. Test if the object implements a "Object" interface 
*)
IF iChObject <> 0 AND_THEN __QUERYINTERFACE(iChObject,iTmp) THEN
	iXpStation := iTmp;
	ToXpStation := TRUE;
END_IF

END_FUNCTION

// COMPONENTs/Optional/Trigger/FB_XP_Trigger
{attribute 'no_explicit_call' := 'Do not call the body - Stick to OOP'}
FUNCTION_BLOCK FB_XP_Trigger EXTENDS FB_CH_Object IMPLEMENTS I_XP_Trigger
VAR
	{attribute 'hide'}
	bInitDone : BOOL;
	{attribute 'hide'}
	ipXpSystem : I_XP_System_Registration;
	{attribute 'hide'}
	ipAccocietedTrack : I_XP_Track;
	{attribute 'hide'}
	ipListOfMoversToCheck : CHALET_BaseComponents.I_CH_LIST;
	{attribute 'hide'}
	fTriggerPositionOnTrack : LREAL;
	{attribute 'hide'}
	eTriggerDirection : Tc3_Mc3Definitions.MC_Direction := Tc3_Mc3Definitions.MC_DIRECTION.mcDirectionPositive;
	{attribute 'hide'}
	ipMoverAtTrigger : I_XP_Mover;
	{attribute 'hide'}
	aMoversPositionLastCycle : ARRAY [0..(CHALET_BaseComponents.BaseParameterlist.MAX_OBJECTS-1)] OF LREAL; // This list is generated at the end of the PRG and contais the positions. The positions are checked in the next cycle
	{attribute 'hide'}
	aMoversTrackLastCycle : ARRAY [0..(CHALET_BaseComponents.BaseParameterlist.MAX_OBJECTS-1)] OF I_XP_Track; // This list is generated at the end of the PRG and contais the track. The tracks are checked in the next cycle
	{attribute 'hide'}
	aMoversInterfaceLastCycle : ARRAY [0..(CHALET_BaseComponents.BaseParameterlist.MAX_OBJECTS-1)] OF I_XP_Mover; // This list is generated at the end of the PRG and contais the Mover interface. The positions are checked in the next cycle
END_VAR

{attribute 'monitoring':='call'}
PROPERTY AccocietedTrack : I_XP_Track
GET
AccocietedTrack := THIS^.ipAccocietedTrack;
END_GET
SET
THIS^.ipAccocietedTrack := AccocietedTrack;
END_SET
END_PROPERTY

METHOD FB_init : BOOL
VAR_INPUT
	bInitRetains : BOOL; // if TRUE, the retain variables are initialized (warm start / cold start)
	bInCopyCode : BOOL;  // if TRUE, the instance afterwards gets moved into the copy code (online change)
	
	ipXpSystem : I_XP_System_Registration; //Interface to XTS system object
	
END_VAR
VAR_INST
	{attribute 'hide'}
	bFBInitCalledOnce : BOOL; //Do the following code once during start up and not during onlinechange
END_VAR
//Do the following code once during start up and not during onlinechange
IF NOT bFBInitCalledOnce THEN 
	;
END_IF

//Regristrate object in System if unknown
IF ipXpSystem <> 0 AND THIS^.ipXpSystem = 0 THEN
	ipXpSystem.RegisterTrigger(THIS^);
	THIS^.ipXpSystem := ipXpSystem;
END_IF

bFBInitCalledOnce := TRUE;
END_METHOD

{attribute 'monitoring':='call'}
PROPERTY HR : HRESULT
GET
IF ipAccocietedTrack <> 0 AND_THEN ipAccocietedTrack.Length > 0 THEN
	HR := S_OK;
ELSE
	HR := E_FAIL;
END_IF
END_GET
END_PROPERTY

METHOD Initialize : HRESULT
IF THIS^.ipXpSystem = 0 THEN
	//No valide interface
	Initialize := E_FAIL;
	RETURN;
END_IF


THIS^.bInitDone := TRUE;
END_METHOD

PROPERTY ListOfMoversToCheck : I_CH_List
SET
IF ListOfMoversToCheck <> 0 THEN
	ipListOfMoversToCheck := ListOfMoversToCheck;
END_IF
END_SET
END_PROPERTY

{attribute 'monitoring':='call'}
PROPERTY MoverAtTrigger : I_XP_Mover
GET
THIS^.Prepare();//Prepare Time-critical information

MoverAtTrigger := ipMoverAtTrigger;
END_GET
END_PROPERTY

{attribute 'monitoring':='call'}
PROPERTY MoverDetected : BOOL
GET
THIS^.Prepare();//Prepare Time-critical information

MoverDetected := (ipMoverAtTrigger <> 0);
END_GET
END_PROPERTY

{attribute 'monitoring':='call'}
PROPERTY PositionOnTrack : LREAL
GET
PositionOnTrack := fTriggerPositionOnTrack;
END_GET
SET
fTriggerPositionOnTrack := PositionOnTrack;
END_SET
END_PROPERTY

(* Time-critical information is processed here, which can then be polled via the property every cycle. 
The update method is usually at the end of the program and then it is already 'outdated'. *)
METHOD PRIVATE Prepare : HRESULT
VAR
	fTrackLentgh : LREAL;
	fMoverActPos,fMoverLastPos : LREAL;
	ipMoverActTrack, ipMoverLastTrack : I_XP_Track;
	fRangePositive, fRangeNegative : LREAL;
	bTriggerIsCloseAtStartTrack, bTriggerIsCloseAtEndTrack : BOOL;
	bMoverWasInRangeNeg, bMoverWasInRangePos, bMoverIsInRangeNeg, bMoverIsInRangePos : BOOL;
	bMoverIsOnSameTrack, bMoverIsOnTrackAhead, bMoverIsOnTrackBehind, bMoverWasOnTrackAhead, bMoverWasOnTrackBehind : BOOL;
	nIdx, nIdxTrack : UDINT;
	fMaxMoveDistPerCycle : LREAL; //[mm] (2 m/s(max. xPlanar speed) * 20ms(max realistic SPS cycle time) + 10%)
END_VAR
VAR_INST
	{attribute 'hide'}
	nLastUpdatedCycleCount : UDINT;
END_VAR
VAR CONSTANT
END_VAR
IF NOT bInitDone OR (THIS^.ipListOfMoversToCheck = 0) OR (THIS^.ipAccocietedTrack = 0) THEN
	Prepare := E_FAIL;
	RETURN;
END_IF

//Check if this Cycle the dates are allready prepared
IF nLastUpdatedCycleCount <> TwinCAT_SystemInfoVarList._TaskInfo[THIS^.nTaskIndex].CycleCount THEN
	nLastUpdatedCycleCount := TwinCAT_SystemInfoVarList._TaskInfo[THIS^.nTaskIndex].CycleCount;
	
	//Abort on invalide interface - Get Track length
	IF ipAccocietedTrack = 0 THEN
		RETURN;
	END_IF
	fTrackLentgh := ipAccocietedTrack.Length;
	
	//Maximum distance a mover can travel in 1 plc cycle. Worstcase 2 m/s(max. xPlanar speed) * 20ms(max realistic SPS cycle time) + 10%
	fMaxMoveDistPerCycle := 2000.0(*2000mm/s=2mm/ms*) * (TwinCAT_SystemInfoVarList._TaskInfo[THIS^.nTaskIndex].CycleTime(*[100ns]*)/10_000)(*CycleTime ms*) / 1000.0 * 1.1(*10%*);
	
	//Clear last stored Mover if an new cycle has started
	THIS^.ipMoverAtTrigger := 0;
	
	//Check old list of Moverspositions and compare them to the current position of the same mover.
	//Set Trigger if the Mover pass the Station
	fRangePositive := MIN((THIS^.fTriggerPositionOnTrack + fMaxMoveDistPerCycle),fTrackLentgh);
	fRangeNegative := MAX((THIS^.fTriggerPositionOnTrack - fMaxMoveDistPerCycle),0); 
	bTriggerIsCloseAtStartTrack := (THIS^.fTriggerPositionOnTrack - fMaxMoveDistPerCycle) < 0.0;
	bTriggerIsCloseAtEndTrack 	:= (THIS^.fTriggerPositionOnTrack + fMaxMoveDistPerCycle) > fTrackLentgh;

		
	FOR nIdx := 0 TO (CHALET_BaseComponents.BaseParameterlist.MAX_OBJECTS-1) DO
		
		IF aMoversInterfaceLastCycle[nIdx] <> 0 THEN
			fMoverActPos 			:= aMoversInterfaceLastCycle[nIdx].PositionOnTrack;
			fMoverLastPos			:= aMoversPositionLastCycle[nIdx];
			ipMoverActTrack 		:= aMoversInterfaceLastCycle[nIdx].CurrentTrack;
			ipMoverLastTrack 		:= aMoversTrackLastCycle[nIdx];
			bMoverIsOnSameTrack 	:= (ipMoverActTrack = ipAccocietedTrack);
			
			//Abort if Lasttrack is not known. Example: first cycle after enabling
			IF ipMoverActTrack = 0 OR ipMoverLastTrack = 0 THEN
				RETURN;
			END_IF
			
			//Reset flags 
			bMoverIsOnTrackAhead 	:= FALSE;		bMoverIsOnTrackBehind 	:= FALSE;		bMoverWasOnTrackAhead 	:= FALSE;		bMoverWasOnTrackBehind 	:= FALSE;
			
			//Test all tracks before and after this track to recognize that the mover has just changed tracks. 
			//This is important if this trigger is near the end or beginning of a track
			FOR nIdxTrack := 0 TO (XPlanarParameterlist.N_MAX_STATIONS_AHEAD_OR_BEHIND-1) DO
				//Tracks Ahead - Mover Is/Was on Track ahead and close(cMaxMoveDistPerCycle) at beginn on track
				IF ipMoverActTrack.TracksStartFromThis[nIdxTrack] <> 0 THEN
					bMoverIsOnTrackAhead 	:= bMoverIsOnTrackAhead 	OR ((ipAccocietedTrack = ipMoverActTrack.TracksStartFromThis[nIdxTrack])  AND ((fMoverActPos - fMaxMoveDistPerCycle) < 0.0));
					bMoverWasOnTrackAhead 	:= bMoverWasOnTrackAhead 	OR ((ipAccocietedTrack = ipMoverLastTrack.TracksStartFromThis[nIdxTrack]) AND ((fMoverLastPos - fMaxMoveDistPerCycle) < 0.0));
				END_IF
				//Tracks Behind - Mover Is/Was on Track behind and close(cMaxMoveDistPerCycle) at end on track
				IF ipMoverActTrack.TracksEndAtThis[nIdxTrack] <> 0 THEN
					bMoverIsOnTrackBehind 	:= bMoverIsOnTrackBehind 	OR ((ipAccocietedTrack = ipMoverActTrack.TracksEndAtThis[nIdxTrack])  AND ((fMoverActPos	+ fMaxMoveDistPerCycle) > ipMoverActTrack.Length));
					bMoverWasOnTrackBehind 	:= bMoverWasOnTrackBehind 	OR ((ipAccocietedTrack = ipMoverLastTrack.TracksEndAtThis[nIdxTrack]) AND ((fMoverLastPos 	+ fMaxMoveDistPerCycle) > ipMoverLastTrack.Length));
				END_IF
			END_FOR
			
			//Closed track and station in close to Modulo pos
			IF bMoverIsOnSameTrack THEN
				bMoverIsOnTrackAhead 	:= ((fMoverActPos - fMaxMoveDistPerCycle) < 0.0);
				bMoverWasOnTrackAhead 	:= ((fMoverLastPos - fMaxMoveDistPerCycle) < 0.0);
				bMoverIsOnTrackBehind 	:= ((fMoverActPos	+ fMaxMoveDistPerCycle) > ipMoverActTrack.Length);
				bMoverWasOnTrackBehind 	:= ((fMoverLastPos 	+ fMaxMoveDistPerCycle) > ipMoverLastTrack.Length);
			END_IF
			
			//Check if Mover passes the station. Ex.: If the Trigger is at Pos 0mm on track, the Mover is never in bRangeNeg. For this case check for bMoverOnTrackBefore
			bMoverIsInRangePos 		:= ((fMoverActPos >= THIS^.fTriggerPositionOnTrack) AND (fMoverActPos <= fRangePositive) AND bMoverIsOnSameTrack) OR (bMoverIsOnTrackAhead 	 AND bTriggerIsCloseAtEndTrack);   
			bMoverIsInRangeNeg 		:= ((fMoverActPos <= THIS^.fTriggerPositionOnTrack) AND (fMoverActPos >= fRangeNegative) AND bMoverIsOnSameTrack) OR (bMoverIsOnTrackBehind  AND bTriggerIsCloseAtStartTrack);     
			bMoverWasInRangePos		:= ((fMoverLastPos > THIS^.fTriggerPositionOnTrack) AND (fMoverLastPos >= fRangeNegative) AND bMoverIsOnSameTrack) OR (bMoverWasOnTrackAhead  AND bTriggerIsCloseAtEndTrack);   
			bMoverWasInRangeNeg		:= ((fMoverLastPos < THIS^.fTriggerPositionOnTrack) AND (fMoverLastPos <= fRangePositive) AND bMoverIsOnSameTrack) OR (bMoverWasOnTrackBehind AND bTriggerIsCloseAtStartTrack);     			

			IF eTriggerDirection = Tc3_Mc3Definitions.MC_DIRECTION.mcDirectionPositive  AND bMoverWasInRangeNeg AND bMoverIsInRangePos AND NOT bMoverWasInRangePos THEN
				THIS^.ipMoverAtTrigger := aMoversInterfaceLastCycle[nIdx];
				RETURN;
			ELSIF eTriggerDirection = Tc3_Mc3Definitions.MC_DIRECTION.mcDirectionNegative AND bMoverIsInRangeNeg AND bMoverWasInRangePos AND NOT bMoverWasInRangeNeg THEN
				THIS^.ipMoverAtTrigger := aMoversInterfaceLastCycle[nIdx];
				RETURN;	
			END_IF
			
		END_IF
	END_FOR
END_IF
END_METHOD

{attribute 'monitoring':='call'}
PROPERTY TimeStamp : Tc2_EtherCAT.T_DCTIME64
GET
THIS^.Prepare();//Prepare Time-critical information

///zzz todo add exact time stamp calculatioin
 IF ipMoverAtTrigger <> 0 THEN
	 TimeStamp := F_GetCurDcTaskTime64();
 ELSE
	 TimeStamp := 0;
 END_IF
END_GET
END_PROPERTY

{attribute 'monitoring':='call'}
PROPERTY TriggerDirection : Tc3_Mc3Definitions.MC_Direction
GET
TriggerDirection := eTriggerDirection;
END_GET
SET
IF TriggerDirection =Tc3_Mc3Definitions.MC_DIRECTION.mcDirectionPositive OR TriggerDirection = Tc3_Mc3Definitions.MC_DIRECTION.mcDirectionNegative THEN
	eTriggerDirection := TriggerDirection;
END_IF
END_SET
END_PROPERTY

METHOD Update : HRESULT
VAR
	nIndex : UINT;
	ipMover : I_XP_Mover;
END_VAR
//Force to do an init befor call update
IF NOT bInitDone THEN
	THIS^.Initialize();
	RETURN;
END_IF

//Clear array
MEMSET(destAddr:=ADR(aMoversInterfaceLastCycle),n:=SIZEOF(aMoversInterfaceLastCycle),fillByte:=0);
MEMSET(destAddr:=ADR(aMoversPositionLastCycle),n:=SIZEOF(aMoversPositionLastCycle),fillByte:=0);
MEMSET(destAddr:=ADR(aMoversTrackLastCycle),n:=SIZEOF(aMoversTrackLastCycle),fillByte:=0);

nIndex := 0;
IF ipListOfMoversToCheck <> 0 THEN
	THIS^.ipListOfMoversToCheck.ResetIterator();
	WHILE THIS^.ipListOfMoversToCheck.HasNextObject() DO
		
		//Cheack all Movers fill the actposition in the array
		IF ToXpMover(THIS^.ipListOfMoversToCheck.GetNextObject(),ipMover) THEN
			aMoversInterfaceLastCycle[nIndex] 	:= ipMover;
			aMoversPositionLastCycle[nIndex] 	:= ipMover.PositionOnTrack;
			aMoversTrackLastCycle[nIndex]		:= ipMover.CurrentTrack;
			nIndex := nIndex +1;
		END_IF
		
	END_WHILE	
	THIS^.ipListOfMoversToCheck.RestoreIterator();
END_IF
END_METHOD

END_FUNCTION_BLOCK

// COMPONENTs/Optional/Trigger/I_XP_Trigger
INTERFACE I_XP_Trigger  EXTENDS __SYSTEM.IQueryInterface

{attribute 'monitoring':='call'}
PROPERTY AccocietedTrack : I_XP_Track
GET
END_GET
SET
END_SET
END_PROPERTY

{attribute 'monitoring':='call'}
PROPERTY HR : HRESULT
GET
END_GET
END_PROPERTY

PROPERTY ListOfMoversToCheck : I_CH_List
SET
END_SET
END_PROPERTY

{attribute 'monitoring':='call'}
PROPERTY MoverAtTrigger : I_XP_Mover
GET
END_GET
END_PROPERTY

{attribute 'monitoring':='call'}
PROPERTY MoverDetected : BOOL
GET
END_GET
END_PROPERTY

{attribute 'monitoring':='call'}
PROPERTY PositionOnTrack : LREAL
GET
END_GET
SET
END_SET
END_PROPERTY

{attribute 'monitoring':='call'}
PROPERTY TimeStamp : T_DCTIME64;
GET
END_GET
END_PROPERTY

{attribute 'monitoring':='call'}
PROPERTY TriggerDirection : Tc3_Mc3Definitions.MC_Direction
GET
END_GET
SET
END_SET
END_PROPERTY

END_INTERFACE

// COMPONENTs/Optional/Zone/FB_XP_SoretedListOfMover
{attribute 'no_explicit_call' := 'Do not call the body - Stick to OOP'}
// Check zone start to end in positive direktion.
FUNCTION_BLOCK FB_XP_SoretedListOfMover EXTENDS FB_CH_Object IMPLEMENTS I_XP_Zone
VAR
	{attribute 'hide'}
	bInitDone : BOOL;
	{attribute 'hide'}
	ipXpStation : I_XP_Station; //Interface to XPlanar station 
	{attribute 'hide'}
	ipListOfMoversToCheck : CHALET_BaseComponents.I_CH_LIST;
	{attribute 'hide'}
	aMoversInZone : ARRAY [0..(CHALET_BaseComponents.BaseParameterlist.MAX_OBJECTS-1)] OF I_XP_Mover_PLC;
END_VAR

{attribute 'monitoring':='call'}
PROPERTY CtsMoversInZone : UINT
GET
VAR
	nIndex : UDINT;
END_VAR
THIS^.Prepare();//Prepare Time-critical information

//Check array for entrys, exit if fisrt empty arrayindex is found.
FOR nIndex := 0 TO (CHALET_BaseComponents.BaseParameterlist.MAX_OBJECTS-1) DO
	IF (aMoversInZone[nIndex] <> 0) THEN
		CtsMoversInZone := CtsMoversInZone +1;
	ELSE
		RETURN;
	END_IF
END_FOR
END_GET
END_PROPERTY

METHOD FB_init : BOOL
VAR_INPUT
	bInitRetains : BOOL; // if TRUE, the retain variables are initialized (warm start / cold start)
	bInCopyCode : BOOL;  // if TRUE, the instance afterwards gets moved into the copy code (online change)
	
	ipXpStation : I_XP_Station; //Interface to XPlanar station 
	ipListOfMoversToCheck : CHALET_BaseComponents.I_CH_LIST;
END_VAR
VAR_INST
	{attribute 'hide'}
	bFBInitCalledOnce : BOOL; //Do the following code once during start up and not during onlinechange
END_VAR
//Do the following code once during start up and not during onlinechange
IF NOT bFBInitCalledOnce THEN 
	;
END_IF

THIS^.ipXpStation := ipXpStation;
THIS^.ipListOfMoversToCheck := ipListOfMoversToCheck;


bFBInitCalledOnce := TRUE;
END_METHOD

METHOD Initialize : HRESULT
IF THIS^.ipXpStation = 0 THEN
	//No valide interface
	Initialize := E_FAIL;
	RETURN;
END_IF

IF THIS^.ipListOfMoversToCheck = 0 THEN
	//No valide interface
	Initialize := E_FAIL;
	RETURN;
END_IF


bInitDone := TRUE;
Initialize := S_OK;
END_METHOD

{attribute 'monitoring':='call'}
// Return a sorted list of movers in this zone. Index 0 is the mover in Front.
PROPERTY MoversInZone : REFERENCE TO ARRAY [0..(CHALET_BaseComponents.BaseParameterlist.MAX_OBJECTS-1)] OF I_XP_Mover_PLC
GET
THIS^.Prepare();//Prepare Time-critical information

MoversInZone REF= THIS^.aMoversInZone;
END_GET
END_PROPERTY

(* Time-critical information is processed here, which can then be polled via the property every cycle. 
The update method is usually at the end of the program and then it is already 'outdated'. *)
METHOD PRIVATE Prepare : HRESULT
VAR
	nLoopIndex : UDINT;
	ipMoverPlc : I_XP_Mover_PLC;
	ipMover : I_XP_Mover;
	ipPath : I_XP_Path;
	fDistToStart : LREAL;
	aDisanceToStart : ARRAY [0..(CHALET_BaseComponents.BaseParameterlist.MAX_OBJECTS-1)] OF LREAL;
END_VAR
VAR_INST
	{attribute 'hide'}
	nLastUpdatedCycleCount : UDINT;
END_VAR
IF NOT bInitDone OR ipXpStation.AccocietedTrack = 0 THEN
	Prepare := E_FAIL;
	RETURN;
END_IF

//Check if this Cycle the dates are allready prepared
IF nLastUpdatedCycleCount <> TwinCAT_SystemInfoVarList._TaskInfo[THIS^.nTaskIndex].CycleCount THEN
	nLastUpdatedCycleCount := TwinCAT_SystemInfoVarList._TaskInfo[THIS^.nTaskIndex].CycleCount;

	//Clear array
	MEMSET(destAddr:=ADR(aMoversInZone),n:=SIZEOF(aMoversInZone),fillByte:=0);
	
	//Cheack all Movers and generate a sorted list of all mover in this zone.
	THIS^.ipListOfMoversToCheck.ResetIterator();
	WHILE THIS^.ipListOfMoversToCheck.HasNextObject() DO
		//Check each mover in this stations list
		IF __QUERYINTERFACE(THIS^.ipListOfMoversToCheck.GetNextObject(),ipMoverPlc) THEN
			
			//mover and distance are known from this point and are now sorted into the array
			fDistToStart := ipMoverPlc.DistToParentStation;
			ipMoverPlc := ipMoverPlc;
			
			//Check array of movers and decide if the current one is closer to 
			FOR nLoopIndex := 0 TO (CHALET_BaseComponents.BaseParameterlist.MAX_OBJECTS-1) DO
				//empty array position
				IF aMoversInZone[nLoopIndex] = 0 THEN
					aMoversInZone[nLoopIndex] := ipMoverPlc;
					aDisanceToStart[nLoopIndex] := fDistToStart;
					EXIT;
					
				//Closer Mover found, move whole array 	
				ELSIF aDisanceToStart[nLoopIndex] > fDistToStart THEN
					MEMMOVE(srcAddr := ADR(aMoversInZone[nLoopIndex]), destAddr := ADR(aMoversInZone[nLoopIndex+1]), n := (SIZEOF(aMoversInZone[0])*(CHALET_BaseComponents.BaseParameterlist.MAX_OBJECTS-1-nLoopIndex)));
					MEMMOVE(srcAddr := ADR(aDisanceToStart[nLoopIndex]), destAddr := ADR(aDisanceToStart[nLoopIndex+1]), n := (SIZEOF(aDisanceToStart[0])*(CHALET_BaseComponents.BaseParameterlist.MAX_OBJECTS-1-nLoopIndex)));
					aMoversInZone[nLoopIndex] := ipMoverPlc;
					aDisanceToStart[nLoopIndex] := fDistToStart;
					EXIT;
					
				//check next position	
				ELSE 
					;
				END_IF
			END_FOR
		END_IF
	END_WHILE
	THIS^.ipListOfMoversToCheck.RestoreIterator();
END_IF
END_METHOD

METHOD Update : HRESULT
VAR

END_VAR
// Nothing.Check Prepare()
END_METHOD

END_FUNCTION_BLOCK

// COMPONENTs/Optional/Zone/I_XP_Zone
INTERFACE I_XP_Zone

{attribute 'monitoring':='call'}
PROPERTY CtsMoversInZone : UINT
GET
END_GET
END_PROPERTY

